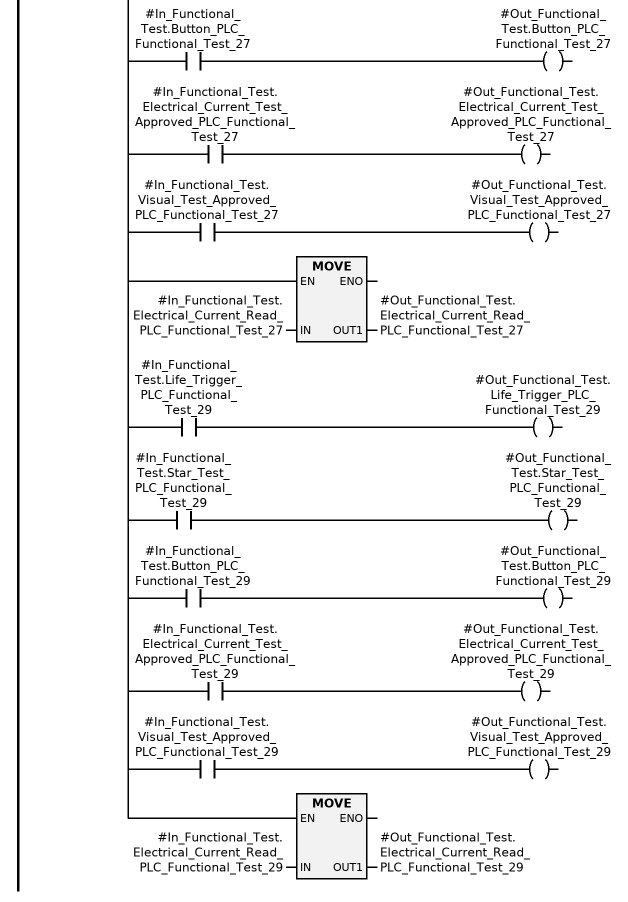
   RUNG wire#powerrail
      { S7_Templates := "SrcType := SInt" } EQ_Contact(in1 := #Test_Station, in2 := 13)
      wire#w1
      Contact( #Life_Trigger )
      Coil( #Out_Functional_Test.Life_Trigger_PLC_Functional_Test_13 )
   END_RUNG
   RUNG wire#w1
      Contact( #Star_Test )
      Coil( #Out_Functional_Test.Star_Test_PLC_Functional_Test_13 )
   END_RUNG
   RUNG wire#w1
      Contact( #Button_Start_Approve )
      Coil( #Out_Functional_Test.Button_PLC_Functional_Test_13 )
   END_RUNG
   RUNG wire#w1
      Contact( #Electrical_Current_Test_Approved )
      Coil( #Out_Functional_Test.Electrical_Current_Test_Approved_PLC_Functional_Test_13 )
   END_RUNG
   RUNG wire#w1
      Contact( #Visual_Test_Approved )
      Coil( #Out_Functional_Test.Visual_Test_Approved_PLC_Functional_Test_13 )
   END_RUNG
   RUNG wire#w1
      Contact( #In_Test_Parameters.Reset_PLC_Functional_Test_13 )
      Coil( #Reset_Functional_Test )
   END_RUNG
   RUNG wire#w1
      Move(in := #Electrical_Current_Read, out1 => #Out_Functional_Test.Electrical_Current_Read_PLC_Functional_Test_13)
   END_RUNG
   RUNG wire#w1
      Contact( #In_Functional_Test.Life_Trigger_PLC_Functional_Test_15 )
      Coil( #Out_Functional_Test.Life_Trigger_PLC_Functional_Test_15 )
   END_RUNG
   RUNG wire#w1
      Contact( #In_Functional_Test.Star_Test_PLC_Functional_Test_15 )
      Coil( #Out_Functional_Test.Star_Test_PLC_Functional_Test_15 )
   END_RUNG
   RUNG wire#w1
      Contact( #In_Functional_Test.Button_PLC_Functional_Test_15 )
      Coil( #Out_Functional_Test.Button_PLC_Functional_Test_15 )
   END_RUNG
   RUNG wire#w1
      Contact( #In_Functional_Test.Electrical_Current_Test_Approved_PLC_Functional_Test_15 )
      Coil( #Out_Functional_Test.Electrical_Current_Test_Approved_PLC_Functional_Test_15 )
   END_RUNG
   RUNG wire#w1
      Contact( #In_Functional_Test.Visual_Test_Approved_PLC_Functional_Test_15 )
      Coil( #Out_Functional_Test.Visual_Test_Approved_PLC_Functional_Test_15 )
   END_RUNG
   RUNG wire#w1
      Move(in := #In_Functional_Test.Electrical_Current_Read_PLC_Functional_Test_15, out1 => #Out_Functional_Test.Electrical_Current_Read_PLC_Functional_Test_15)
   END_RUNG
   RUNG wire#w1
      Contact( #In_Functional_Test.Life_Trigger_PLC_Functional_Test_17 )
      Coil( #Out_Functional_Test.Life_Trigger_PLC_Functional_Test_17 )
   END_RUNG
   RUNG wire#w1
      Contact( #In_Functional_Test.Star_Test_PLC_Functional_Test_17 )
      Coil( #Out_Functional_Test.Star_Test_PLC_Functional_Test_17 )
   END_RUNG
   RUNG wire#w1
      Contact( #In_Functional_Test.Button_PLC_Functional_Test_17 )
      Coil( #Out_Functional_Test.Button_PLC_Functional_Test_17 )
   END_RUNG
   RUNG wire#w1
      Contact( #In_Functional_Test.Electrical_Current_Test_Approved_PLC_Functional_Test_17 )
      Coil( #Out_Functional_Test.Electrical_Current_Test_Approved_PLC_Functional_Test_17 )
   END_RUNG
   RUNG wire#w1
      Contact( #In_Functional_Test.Visual_Test_Approved_PLC_Functional_Test_17 )
      Coil( #Out_Functional_Test.Visual_Test_Approved_PLC_Functional_Test_17 )
   END_RUNG
   RUNG wire#w1
      Move(in := #In_Functional_Test.Electrical_Current_Read_PLC_Functional_Test_17, out1 => #Out_Functional_Test.Electrical_Current_Read_PLC_Functional_Test_17)
   END_RUNG
   RUNG wire#w1
      Contact( #In_Functional_Test.Life_Trigger_PLC_Functional_Test_19 )
      Coil( #Out_Functional_Test.Life_Trigger_PLC_Functional_Test_19 )
   END_RUNG
   RUNG wire#w1
      Contact( #In_Functional_Test.Star_Test_PLC_Functional_Test_19 )
      Coil( #Out_Functional_Test.Star_Test_PLC_Functional_Test_19 )
   END_RUNG
   RUNG wire#w1
      Contact( #In_Functional_Test.Button_PLC_Functional_Test_19 )
      Coil( #Out_Functional_Test.Button_PLC_Functional_Test_19 )
   END_RUNG
   RUNG wire#w1
      Contact( #In_Functional_Test.Electrical_Current_Test_Approved_PLC_Functional_Test_19 )
      Coil( #Out_Functional_Test.Electrical_Current_Test_Approved_PLC_Functional_Test_19 )
   END_RUNG
   RUNG wire#w1
      Contact( #In_Functional_Test.Visual_Test_Approved_PLC_Functional_Test_19 )
      Coil( #Out_Functional_Test.Visual_Test_Approved_PLC_Functional_Test_19 )
   END_RUNG
   RUNG wire#w1
      Move(in := #In_Functional_Test.Electrical_Current_Read_PLC_Functional_Test_19, out1 => #Out_Functional_Test.Electrical_Current_Read_PLC_Functional_Test_19)
   END_RUNG
   RUNG wire#w1
      Contact( #In_Functional_Test.Life_Trigger_PLC_Functional_Test_21 )
      Coil( #Out_Functional_Test.Life_Trigger_PLC_Functional_Test_21 )
   END_RUNG
   RUNG wire#w1
      Contact( #In_Functional_Test.Star_Test_PLC_Functional_Test_21 )
      Coil( #Out_Functional_Test.Star_Test_PLC_Functional_Test_21 )
   END_RUNG
   RUNG wire#w1
      Contact( #In_Functional_Test.Button_PLC_Functional_Test_21 )
      Coil( #Out_Functional_Test.Button_PLC_Functional_Test_21 )
   END_RUNG
   RUNG wire#w1
      Contact( #In_Functional_Test.Electrical_Current_Test_Approved_PLC_Functional_Test_21 )
      Coil( #Out_Functional_Test.Electrical_Current_Test_Approved_PLC_Functional_Test_21 )
   END_RUNG
   RUNG wire#w1
      Contact( #In_Functional_Test.Visual_Test_Approved_PLC_Functional_Test_21 )
      Coil( #Out_Functional_Test.Visual_Test_Approved_PLC_Functional_Test_21 )
   END_RUNG
   RUNG wire#w1
      Move(in := #In_Functional_Test.Electrical_Current_Read_PLC_Functional_Test_21, out1 => #Out_Functional_Test.Electrical_Current_Read_PLC_Functional_Test_21)
   END_RUNG
   RUNG wire#w1
      Contact( #In_Functional_Test.Life_Trigger_PLC_Functional_Test_23 )
      Coil( #Out_Functional_Test.Life_Trigger_PLC_Functional_Test_23 )
   END_RUNG
   RUNG wire#w1
      Contact( #In_Functional_Test.Star_Test_PLC_Functional_Test_23 )
      Coil( #Out_Functional_Test.Star_Test_PLC_Functional_Test_23 )
   END_RUNG
   RUNG wire#w1
      Contact( #In_Functional_Test.Button_PLC_Functional_Test_23 )
      Coil( #Out_Functional_Test.Button_PLC_Functional_Test_23 )
   END_RUNG
   RUNG wire#w1
      Contact( #In_Functional_Test.Electrical_Current_Test_Approved_PLC_Functional_Test_23 )
      Coil( #Out_Functional_Test.Electrical_Current_Test_Approved_PLC_Functional_Test_23 )
   END_RUNG
   RUNG wire#w1
      Contact( #In_Functional_Test.Visual_Test_Approved_PLC_Functional_Test_23 )
      Coil( #Out_Functional_Test.Visual_Test_Approved_PLC_Functional_Test_23 )
   END_RUNG
   RUNG wire#w1
      Move(in := #In_Functional_Test.Electrical_Current_Read_PLC_Functional_Test_23, out1 => #Out_Functional_Test.Electrical_Current_Read_PLC_Functional_Test_23)
   END_RUNG
   RUNG wire#w1
      Contact( #In_Functional_Test.Life_Trigger_PLC_Functional_Test_25 )
      Coil( #Out_Functional_Test.Life_Trigger_PLC_Functional_Test_25 )
   END_RUNG
   RUNG wire#w1
      Contact( #In_Functional_Test.Star_Test_PLC_Functional_Test_25 )
      Coil( #Out_Functional_Test.Star_Test_PLC_Functional_Test_25 )
   END_RUNG
   RUNG wire#w1
      Contact( #In_Functional_Test.Button_PLC_Functional_Test_25 )
      Coil( #Out_Functional_Test.Button_PLC_Functional_Test_25 )
   END_RUNG
   RUNG wire#w1
      Contact( #In_Functional_Test.Electrical_Current_Test_Approved_PLC_Functional_Test_25 )
      Coil( #Out_Functional_Test.Electrical_Current_Test_Approved_PLC_Functional_Test_25 )
   END_RUNG
   RUNG wire#w1
      Contact( #In_Functional_Test.Visual_Test_Approved_PLC_Functional_Test_25 )
      Coil( #Out_Functional_Test.Visual_Test_Approved_PLC_Functional_Test_25 )
   END_RUNG
   RUNG wire#w1
      Move(in := #In_Functional_Test.Electrical_Current_Read_PLC_Functional_Test_25, out1 => #Out_Functional_Test.Electrical_Current_Read_PLC_Functional_Test_25)
   END_RUNG
   RUNG wire#w1
      Contact( #In_Functional_Test.Life_Trigger_PLC_Functional_Test_27 )
      Coil( #Out_Functional_Test.Life_Trigger_PLC_Functional_Test_27 )
   END_RUNG
   RUNG wire#w1
      Contact( #In_Functional_Test.Star_Test_PLC_Functional_Test_27 )
      Coil( #Out_Functional_Test.Star_Test_PLC_Functional_Test_27 )
   END_RUNG
   RUNG wire#w1
      Contact( #In_Functional_Test.Button_PLC_Functional_Test_27 )
      Coil( #Out_Functional_Test.Button_PLC_Functional_Test_27 )
   END_RUNG
   RUNG wire#w1
      Contact( #In_Functional_Test.Electrical_Current_Test_Approved_PLC_Functional_Test_27 )
      Coil( #Out_Functional_Test.Electrical_Current_Test_Approved_PLC_Functional_Test_27 )
   END_RUNG
   RUNG wire#w1
      Contact( #In_Functional_Test.Visual_Test_Approved_PLC_Functional_Test_27 )
      Coil( #Out_Functional_Test.Visual_Test_Approved_PLC_Functional_Test_27 )
   END_RUNG
   RUNG wire#w1
      Move(in := #In_Functional_Test.Electrical_Current_Read_PLC_Functional_Test_27, out1 => #Out_Functional_Test.Electrical_Current_Read_PLC_Functional_Test_27)
   END_RUNG
   RUNG wire#w1
      Contact( #In_Functional_Test.Life_Trigger_PLC_Functional_Test_29 )
      Coil( #Out_Functional_Test.Life_Trigger_PLC_Functional_Test_29 )
   END_RUNG
   RUNG wire#w1
      Contact( #In_Functional_Test.Star_Test_PLC_Functional_Test_29 )
      Coil( #Out_Functional_Test.Star_Test_PLC_Functional_Test_29 )
   END_RUNG
   RUNG wire#w1
      Contact( #In_Functional_Test.Button_PLC_Functional_Test_29 )
      Coil( #Out_Functional_Test.Button_PLC_Functional_Test_29 )
   END_RUNG
   RUNG wire#w1
      Contact( #In_Functional_Test.Electrical_Current_Test_Approved_PLC_Functional_Test_29 )
      Coil( #Out_Functional_Test.Electrical_Current_Test_Approved_PLC_Functional_Test_29 )
   END_RUNG
   RUNG wire#w1
      Contact( #In_Functional_Test.Visual_Test_Approved_PLC_Functional_Test_29 )
      Coil( #Out_Functional_Test.Visual_Test_Approved_PLC_Functional_Test_29 )
   END_RUNG
   RUNG wire#w1
      Move(in := #In_Functional_Test.Electrical_Current_Read_PLC_Functional_Test_29, out1 => #Out_Functional_Test.Electrical_Current_Read_PLC_Functional_Test_29)
   END_RUNG
   // the same network as SCL:
   #_w1 := #Test_Station = 13;
   #Out_Functional_Test.Life_Trigger_PLC_Functional_Test_13 := #_w1 AND #Life_Trigger;
   #Out_Functional_Test.Star_Test_PLC_Functional_Test_13 := #_w1 AND #Star_Test;
   #Out_Functional_Test.Button_PLC_Functional_Test_13 := #_w1 AND #Button_Start_Approve;
   #Out_Functional_Test.Electrical_Current_Test_Approved_PLC_Functional_Test_13 := #_w1 AND #Electrical_Current_Test_Approved;
   #Out_Functional_Test.Visual_Test_Approved_PLC_Functional_Test_13 := #_w1 AND #Visual_Test_Approved;
   #Reset_Functional_Test := #_w1 AND #In_Test_Parameters.Reset_PLC_Functional_Test_13;
   IF #_w1 THEN
       #Out_Functional_Test.Electrical_Current_Read_PLC_Functional_Test_13 := #Electrical_Current_Read;
   END_IF;
   #Out_Functional_Test.Life_Trigger_PLC_Functional_Test_15 := #_w1 AND #In_Functional_Test.Life_Trigger_PLC_Functional_Test_15;
   #Out_Functional_Test.Star_Test_PLC_Functional_Test_15 := #_w1 AND #In_Functional_Test.Star_Test_PLC_Functional_Test_15;
   #Out_Functional_Test.Button_PLC_Functional_Test_15 := #_w1 AND #In_Functional_Test.Button_PLC_Functional_Test_15;
   #Out_Functional_Test.Electrical_Current_Test_Approved_PLC_Functional_Test_15 := #_w1 AND #In_Functional_Test.Electrical_Current_Test_Approved_PLC_Functional_Test_15;
   #Out_Functional_Test.Visual_Test_Approved_PLC_Functional_Test_15 := #_w1 AND #In_Functional_Test.Visual_Test_Approved_PLC_Functional_Test_15;
   IF #_w1 THEN
       #Out_Functional_Test.Electrical_Current_Read_PLC_Functional_Test_15 := #In_Functional_Test.Electrical_Current_Read_PLC_Functional_Test_15;
   END_IF;
   #Out_Functional_Test.Life_Trigger_PLC_Functional_Test_17 := #_w1 AND #In_Functional_Test.Life_Trigger_PLC_Functional_Test_17;
   #Out_Functional_Test.Star_Test_PLC_Functional_Test_17 := #_w1 AND #In_Functional_Test.Star_Test_PLC_Functional_Test_17;
   #Out_Functional_Test.Button_PLC_Functional_Test_17 := #_w1 AND #In_Functional_Test.Button_PLC_Functional_Test_17;
   #Out_Functional_Test.Electrical_Current_Test_Approved_PLC_Functional_Test_17 := #_w1 AND #In_Functional_Test.Electrical_Current_Test_Approved_PLC_Functional_Test_17;
   #Out_Functional_Test.Visual_Test_Approved_PLC_Functional_Test_17 := #_w1 AND #In_Functional_Test.Visual_Test_Approved_PLC_Functional_Test_17;
   IF #_w1 THEN
       #Out_Functional_Test.Electrical_Current_Read_PLC_Functional_Test_17 := #In_Functional_Test.Electrical_Current_Read_PLC_Functional_Test_17;
   END_IF;
   #Out_Functional_Test.Life_Trigger_PLC_Functional_Test_19 := #_w1 AND #In_Functional_Test.Life_Trigger_PLC_Functional_Test_19;
   #Out_Functional_Test.Star_Test_PLC_Functional_Test_19 := #_w1 AND #In_Functional_Test.Star_Test_PLC_Functional_Test_19;
   #Out_Functional_Test.Button_PLC_Functional_Test_19 := #_w1 AND #In_Functional_Test.Button_PLC_Functional_Test_19;
   #Out_Functional_Test.Electrical_Current_Test_Approved_PLC_Functional_Test_19 := #_w1 AND #In_Functional_Test.Electrical_Current_Test_Approved_PLC_Functional_Test_19;
   #Out_Functional_Test.Visual_Test_Approved_PLC_Functional_Test_19 := #_w1 AND #In_Functional_Test.Visual_Test_Approved_PLC_Functional_Test_19;
   IF #_w1 THEN
       #Out_Functional_Test.Electrical_Current_Read_PLC_Functional_Test_19 := #In_Functional_Test.Electrical_Current_Read_PLC_Functional_Test_19;
   END_IF;
   #Out_Functional_Test.Life_Trigger_PLC_Functional_Test_21 := #_w1 AND #In_Functional_Test.Life_Trigger_PLC_Functional_Test_21;
   #Out_Functional_Test.Star_Test_PLC_Functional_Test_21 := #_w1 AND #In_Functional_Test.Star_Test_PLC_Functional_Test_21;
   #Out_Functional_Test.Button_PLC_Functional_Test_21 := #_w1 AND #In_Functional_Test.Button_PLC_Functional_Test_21;
   #Out_Functional_Test.Electrical_Current_Test_Approved_PLC_Functional_Test_21 := #_w1 AND #In_Functional_Test.Electrical_Current_Test_Approved_PLC_Functional_Test_21;
   #Out_Functional_Test.Visual_Test_Approved_PLC_Functional_Test_21 := #_w1 AND #In_Functional_Test.Visual_Test_Approved_PLC_Functional_Test_21;
   IF #_w1 THEN
       #Out_Functional_Test.Electrical_Current_Read_PLC_Functional_Test_21 := #In_Functional_Test.Electrical_Current_Read_PLC_Functional_Test_21;
   END_IF;
   #Out_Functional_Test.Life_Trigger_PLC_Functional_Test_23 := #_w1 AND #In_Functional_Test.Life_Trigger_PLC_Functional_Test_23;
   #Out_Functional_Test.Star_Test_PLC_Functional_Test_23 := #_w1 AND #In_Functional_Test.Star_Test_PLC_Functional_Test_23;
   #Out_Functional_Test.Button_PLC_Functional_Test_23 := #_w1 AND #In_Functional_Test.Button_PLC_Functional_Test_23;
   #Out_Functional_Test.Electrical_Current_Test_Approved_PLC_Functional_Test_23 := #_w1 AND #In_Functional_Test.Electrical_Current_Test_Approved_PLC_Functional_Test_23;
   #Out_Functional_Test.Visual_Test_Approved_PLC_Functional_Test_23 := #_w1 AND #In_Functional_Test.Visual_Test_Approved_PLC_Functional_Test_23;
   IF #_w1 THEN
       #Out_Functional_Test.Electrical_Current_Read_PLC_Functional_Test_23 := #In_Functional_Test.Electrical_Current_Read_PLC_Functional_Test_23;
   END_IF;
   #Out_Functional_Test.Life_Trigger_PLC_Functional_Test_25 := #_w1 AND #In_Functional_Test.Life_Trigger_PLC_Functional_Test_25;
   #Out_Functional_Test.Star_Test_PLC_Functional_Test_25 := #_w1 AND #In_Functional_Test.Star_Test_PLC_Functional_Test_25;
   #Out_Functional_Test.Button_PLC_Functional_Test_25 := #_w1 AND #In_Functional_Test.Button_PLC_Functional_Test_25;
   #Out_Functional_Test.Electrical_Current_Test_Approved_PLC_Functional_Test_25 := #_w1 AND #In_Functional_Test.Electrical_Current_Test_Approved_PLC_Functional_Test_25;
   #Out_Functional_Test.Visual_Test_Approved_PLC_Functional_Test_25 := #_w1 AND #In_Functional_Test.Visual_Test_Approved_PLC_Functional_Test_25;
   IF #_w1 THEN
       #Out_Functional_Test.Electrical_Current_Read_PLC_Functional_Test_25 := #In_Functional_Test.Electrical_Current_Read_PLC_Functional_Test_25;
   END_IF;
   #Out_Functional_Test.Life_Trigger_PLC_Functional_Test_27 := #_w1 AND #In_Functional_Test.Life_Trigger_PLC_Functional_Test_27;
   #Out_Functional_Test.Star_Test_PLC_Functional_Test_27 := #_w1 AND #In_Functional_Test.Star_Test_PLC_Functional_Test_27;
   #Out_Functional_Test.Button_PLC_Functional_Test_27 := #_w1 AND #In_Functional_Test.Button_PLC_Functional_Test_27;
   #Out_Functional_Test.Electrical_Current_Test_Approved_PLC_Functional_Test_27 := #_w1 AND #In_Functional_Test.Electrical_Current_Test_Approved_PLC_Functional_Test_27;
   #Out_Functional_Test.Visual_Test_Approved_PLC_Functional_Test_27 := #_w1 AND #In_Functional_Test.Visual_Test_Approved_PLC_Functional_Test_27;
   IF #_w1 THEN
       #Out_Functional_Test.Electrical_Current_Read_PLC_Functional_Test_27 := #In_Functional_Test.Electrical_Current_Read_PLC_Functional_Test_27;
   END_IF;
   #Out_Functional_Test.Life_Trigger_PLC_Functional_Test_29 := #_w1 AND #In_Functional_Test.Life_Trigger_PLC_Functional_Test_29;
   #Out_Functional_Test.Star_Test_PLC_Functional_Test_29 := #_w1 AND #In_Functional_Test.Star_Test_PLC_Functional_Test_29;
   #Out_Functional_Test.Button_PLC_Functional_Test_29 := #_w1 AND #In_Functional_Test.Button_PLC_Functional_Test_29;
   #Out_Functional_Test.Electrical_Current_Test_Approved_PLC_Functional_Test_29 := #_w1 AND #In_Functional_Test.Electrical_Current_Test_Approved_PLC_Functional_Test_29;
   #Out_Functional_Test.Visual_Test_Approved_PLC_Functional_Test_29 := #_w1 AND #In_Functional_Test.Visual_Test_Approved_PLC_Functional_Test_29;
   IF #_w1 THEN
       #Out_Functional_Test.Electrical_Current_Read_PLC_Functional_Test_29 := #In_Functional_Test.Electrical_Current_Read_PLC_Functional_Test_29;
   END_IF;
END_REGION

REGION Network 9: Functional Test Station 15
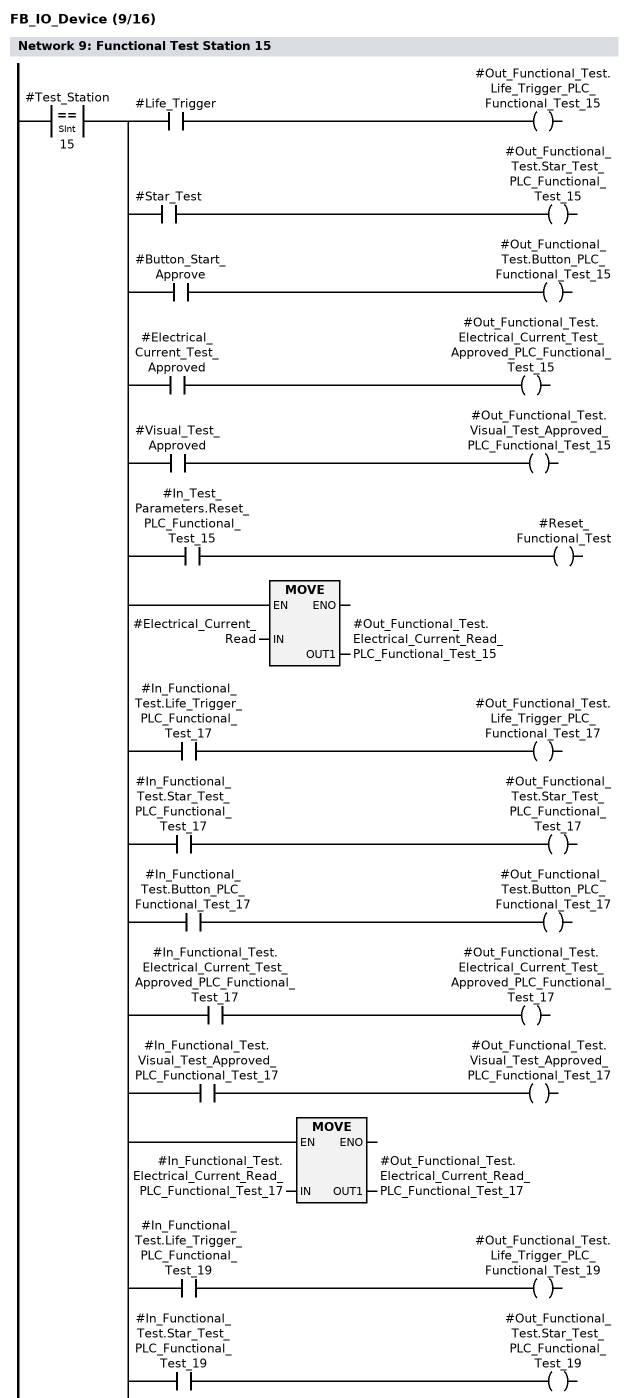
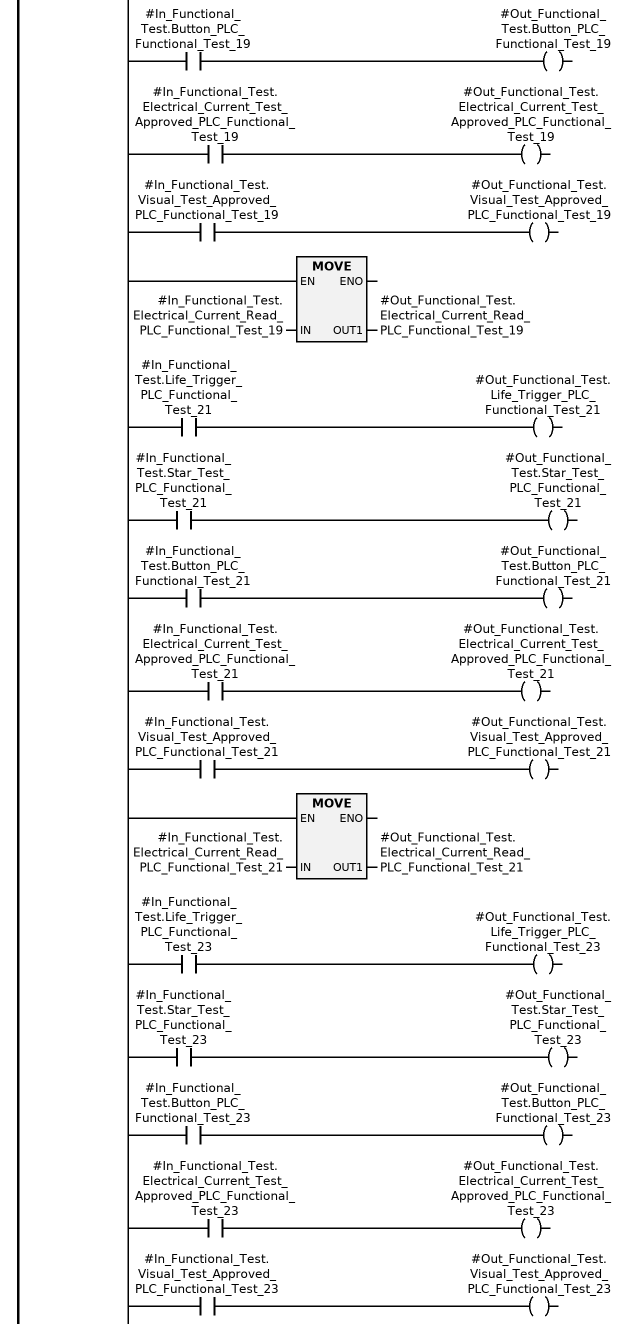
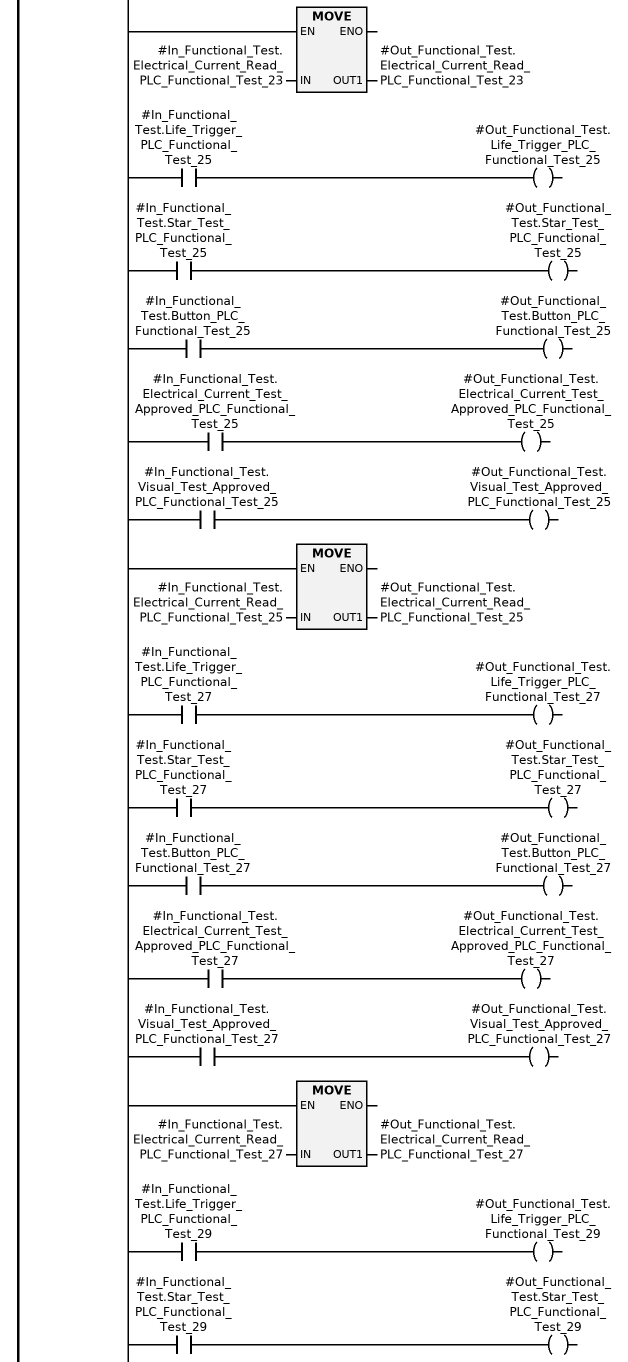
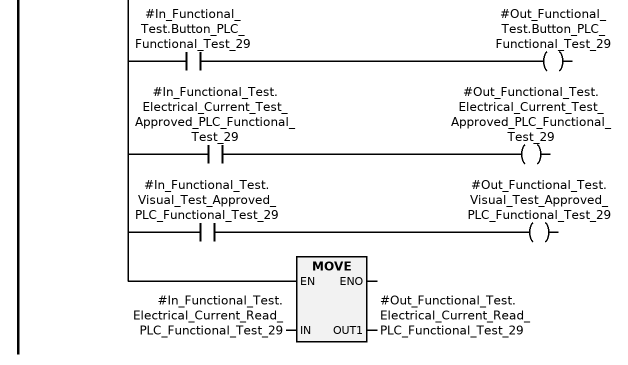
   RUNG wire#powerrail
      { S7_Templates := "SrcType := SInt" } EQ_Contact(in1 := #Test_Station, in2 := 15)
      wire#w1
      Contact( #Life_Trigger )
      Coil( #Out_Functional_Test.Life_Trigger_PLC_Functional_Test_15 )
   END_RUNG
   RUNG wire#w1
      Contact( #Star_Test )
      Coil( #Out_Functional_Test.Star_Test_PLC_Functional_Test_15 )
   END_RUNG
   RUNG wire#w1
      Contact( #Button_Start_Approve )
      Coil( #Out_Functional_Test.Button_PLC_Functional_Test_15 )
   END_RUNG
   RUNG wire#w1
      Contact( #Electrical_Current_Test_Approved )
      Coil( #Out_Functional_Test.Electrical_Current_Test_Approved_PLC_Functional_Test_15 )
   END_RUNG
   RUNG wire#w1
      Contact( #Visual_Test_Approved )
      Coil( #Out_Functional_Test.Visual_Test_Approved_PLC_Functional_Test_15 )
   END_RUNG
   RUNG wire#w1
      Contact( #In_Test_Parameters.Reset_PLC_Functional_Test_15 )
      Coil( #Reset_Functional_Test )
   END_RUNG
   RUNG wire#w1
      Move(in := #Electrical_Current_Read, out1 => #Out_Functional_Test.Electrical_Current_Read_PLC_Functional_Test_15)
   END_RUNG
   RUNG wire#w1
      Contact( #In_Functional_Test.Life_Trigger_PLC_Functional_Test_17 )
      Coil( #Out_Functional_Test.Life_Trigger_PLC_Functional_Test_17 )
   END_RUNG
   RUNG wire#w1
      Contact( #In_Functional_Test.Star_Test_PLC_Functional_Test_17 )
      Coil( #Out_Functional_Test.Star_Test_PLC_Functional_Test_17 )
   END_RUNG
   RUNG wire#w1
      Contact( #In_Functional_Test.Button_PLC_Functional_Test_17 )
      Coil( #Out_Functional_Test.Button_PLC_Functional_Test_17 )
   END_RUNG
   RUNG wire#w1
      Contact( #In_Functional_Test.Electrical_Current_Test_Approved_PLC_Functional_Test_17 )
      Coil( #Out_Functional_Test.Electrical_Current_Test_Approved_PLC_Functional_Test_17 )
   END_RUNG
   RUNG wire#w1
      Contact( #In_Functional_Test.Visual_Test_Approved_PLC_Functional_Test_17 )
      Coil( #Out_Functional_Test.Visual_Test_Approved_PLC_Functional_Test_17 )
   END_RUNG
   RUNG wire#w1
      Move(in := #In_Functional_Test.Electrical_Current_Read_PLC_Functional_Test_17, out1 => #Out_Functional_Test.Electrical_Current_Read_PLC_Functional_Test_17)
   END_RUNG
   RUNG wire#w1
      Contact( #In_Functional_Test.Life_Trigger_PLC_Functional_Test_19 )
      Coil( #Out_Functional_Test.Life_Trigger_PLC_Functional_Test_19 )
   END_RUNG
   RUNG wire#w1
      Contact( #In_Functional_Test.Star_Test_PLC_Functional_Test_19 )
      Coil( #Out_Functional_Test.Star_Test_PLC_Functional_Test_19 )
   END_RUNG
   RUNG wire#w1
      Contact( #In_Functional_Test.Button_PLC_Functional_Test_19 )
      Coil( #Out_Functional_Test.Button_PLC_Functional_Test_19 )
   END_RUNG
   RUNG wire#w1
      Contact( #In_Functional_Test.Electrical_Current_Test_Approved_PLC_Functional_Test_19 )
      Coil( #Out_Functional_Test.Electrical_Current_Test_Approved_PLC_Functional_Test_19 )
   END_RUNG
   RUNG wire#w1
      Contact( #In_Functional_Test.Visual_Test_Approved_PLC_Functional_Test_19 )
      Coil( #Out_Functional_Test.Visual_Test_Approved_PLC_Functional_Test_19 )
   END_RUNG
   RUNG wire#w1
      Move(in := #In_Functional_Test.Electrical_Current_Read_PLC_Functional_Test_19, out1 => #Out_Functional_Test.Electrical_Current_Read_PLC_Functional_Test_19)
   END_RUNG
   RUNG wire#w1
      Contact( #In_Functional_Test.Life_Trigger_PLC_Functional_Test_21 )
      Coil( #Out_Functional_Test.Life_Trigger_PLC_Functional_Test_21 )
   END_RUNG
   RUNG wire#w1
      Contact( #In_Functional_Test.Star_Test_PLC_Functional_Test_21 )
      Coil( #Out_Functional_Test.Star_Test_PLC_Functional_Test_21 )
   END_RUNG
   RUNG wire#w1
      Contact( #In_Functional_Test.Button_PLC_Functional_Test_21 )
      Coil( #Out_Functional_Test.Button_PLC_Functional_Test_21 )
   END_RUNG
   RUNG wire#w1
      Contact( #In_Functional_Test.Electrical_Current_Test_Approved_PLC_Functional_Test_21 )
      Coil( #Out_Functional_Test.Electrical_Current_Test_Approved_PLC_Functional_Test_21 )
   END_RUNG
   RUNG wire#w1
      Contact( #In_Functional_Test.Visual_Test_Approved_PLC_Functional_Test_21 )
      Coil( #Out_Functional_Test.Visual_Test_Approved_PLC_Functional_Test_21 )
   END_RUNG
   RUNG wire#w1
      Move(in := #In_Functional_Test.Electrical_Current_Read_PLC_Functional_Test_21, out1 => #Out_Functional_Test.Electrical_Current_Read_PLC_Functional_Test_21)
   END_RUNG
   RUNG wire#w1
      Contact( #In_Functional_Test.Life_Trigger_PLC_Functional_Test_23 )
      Coil( #Out_Functional_Test.Life_Trigger_PLC_Functional_Test_23 )
   END_RUNG
   RUNG wire#w1
      Contact( #In_Functional_Test.Star_Test_PLC_Functional_Test_23 )
      Coil( #Out_Functional_Test.Star_Test_PLC_Functional_Test_23 )
   END_RUNG
   RUNG wire#w1
      Contact( #In_Functional_Test.Button_PLC_Functional_Test_23 )
      Coil( #Out_Functional_Test.Button_PLC_Functional_Test_23 )
   END_RUNG
   RUNG wire#w1
      Contact( #In_Functional_Test.Electrical_Current_Test_Approved_PLC_Functional_Test_23 )
      Coil( #Out_Functional_Test.Electrical_Current_Test_Approved_PLC_Functional_Test_23 )
   END_RUNG
   RUNG wire#w1
      Contact( #In_Functional_Test.Visual_Test_Approved_PLC_Functional_Test_23 )
      Coil( #Out_Functional_Test.Visual_Test_Approved_PLC_Functional_Test_23 )
   END_RUNG
   RUNG wire#w1
      Move(in := #In_Functional_Test.Electrical_Current_Read_PLC_Functional_Test_23, out1 => #Out_Functional_Test.Electrical_Current_Read_PLC_Functional_Test_23)
   END_RUNG
   RUNG wire#w1
      Contact( #In_Functional_Test.Life_Trigger_PLC_Functional_Test_25 )
      Coil( #Out_Functional_Test.Life_Trigger_PLC_Functional_Test_25 )
   END_RUNG
   RUNG wire#w1
      Contact( #In_Functional_Test.Star_Test_PLC_Functional_Test_25 )
      Coil( #Out_Functional_Test.Star_Test_PLC_Functional_Test_25 )
   END_RUNG
   RUNG wire#w1
      Contact( #In_Functional_Test.Button_PLC_Functional_Test_25 )
      Coil( #Out_Functional_Test.Button_PLC_Functional_Test_25 )
   END_RUNG
   RUNG wire#w1
      Contact( #In_Functional_Test.Electrical_Current_Test_Approved_PLC_Functional_Test_25 )
      Coil( #Out_Functional_Test.Electrical_Current_Test_Approved_PLC_Functional_Test_25 )
   END_RUNG
   RUNG wire#w1
      Contact( #In_Functional_Test.Visual_Test_Approved_PLC_Functional_Test_25 )
      Coil( #Out_Functional_Test.Visual_Test_Approved_PLC_Functional_Test_25 )
   END_RUNG
   RUNG wire#w1
      Move(in := #In_Functional_Test.Electrical_Current_Read_PLC_Functional_Test_25, out1 => #Out_Functional_Test.Electrical_Current_Read_PLC_Functional_Test_25)
   END_RUNG
   RUNG wire#w1
      Contact( #In_Functional_Test.Life_Trigger_PLC_Functional_Test_27 )
      Coil( #Out_Functional_Test.Life_Trigger_PLC_Functional_Test_27 )
   END_RUNG
   RUNG wire#w1
      Contact( #In_Functional_Test.Star_Test_PLC_Functional_Test_27 )
      Coil( #Out_Functional_Test.Star_Test_PLC_Functional_Test_27 )
   END_RUNG
   RUNG wire#w1
      Contact( #In_Functional_Test.Button_PLC_Functional_Test_27 )
      Coil( #Out_Functional_Test.Button_PLC_Functional_Test_27 )
   END_RUNG
   RUNG wire#w1
      Contact( #In_Functional_Test.Electrical_Current_Test_Approved_PLC_Functional_Test_27 )
      Coil( #Out_Functional_Test.Electrical_Current_Test_Approved_PLC_Functional_Test_27 )
   END_RUNG
   RUNG wire#w1
      Contact( #In_Functional_Test.Visual_Test_Approved_PLC_Functional_Test_27 )
      Coil( #Out_Functional_Test.Visual_Test_Approved_PLC_Functional_Test_27 )
   END_RUNG
   RUNG wire#w1
      Move(in := #In_Functional_Test.Electrical_Current_Read_PLC_Functional_Test_27, out1 => #Out_Functional_Test.Electrical_Current_Read_PLC_Functional_Test_27)
   END_RUNG
   RUNG wire#w1
      Contact( #In_Functional_Test.Life_Trigger_PLC_Functional_Test_29 )
      Coil( #Out_Functional_Test.Life_Trigger_PLC_Functional_Test_29 )
   END_RUNG
   RUNG wire#w1
      Contact( #In_Functional_Test.Star_Test_PLC_Functional_Test_29 )
      Coil( #Out_Functional_Test.Star_Test_PLC_Functional_Test_29 )
   END_RUNG
   RUNG wire#w1
      Contact( #In_Functional_Test.Button_PLC_Functional_Test_29 )
      Coil( #Out_Functional_Test.Button_PLC_Functional_Test_29 )
   END_RUNG
   RUNG wire#w1
      Contact( #In_Functional_Test.Electrical_Current_Test_Approved_PLC_Functional_Test_29 )
      Coil( #Out_Functional_Test.Electrical_Current_Test_Approved_PLC_Functional_Test_29 )
   END_RUNG
   RUNG wire#w1
      Contact( #In_Functional_Test.Visual_Test_Approved_PLC_Functional_Test_29 )
      Coil( #Out_Functional_Test.Visual_Test_Approved_PLC_Functional_Test_29 )
   END_RUNG
   RUNG wire#w1
      Move(in := #In_Functional_Test.Electrical_Current_Read_PLC_Functional_Test_29, out1 => #Out_Functional_Test.Electrical_Current_Read_PLC_Functional_Test_29)
   END_RUNG
   // the same network as SCL:
   #_w1 := #Test_Station = 15;
   #Out_Functional_Test.Life_Trigger_PLC_Functional_Test_15 := #_w1 AND #Life_Trigger;
   #Out_Functional_Test.Star_Test_PLC_Functional_Test_15 := #_w1 AND #Star_Test;
   #Out_Functional_Test.Button_PLC_Functional_Test_15 := #_w1 AND #Button_Start_Approve;
   #Out_Functional_Test.Electrical_Current_Test_Approved_PLC_Functional_Test_15 := #_w1 AND #Electrical_Current_Test_Approved;
   #Out_Functional_Test.Visual_Test_Approved_PLC_Functional_Test_15 := #_w1 AND #Visual_Test_Approved;
   #Reset_Functional_Test := #_w1 AND #In_Test_Parameters.Reset_PLC_Functional_Test_15;
   IF #_w1 THEN
       #Out_Functional_Test.Electrical_Current_Read_PLC_Functional_Test_15 := #Electrical_Current_Read;
   END_IF;
   #Out_Functional_Test.Life_Trigger_PLC_Functional_Test_17 := #_w1 AND #In_Functional_Test.Life_Trigger_PLC_Functional_Test_17;
   #Out_Functional_Test.Star_Test_PLC_Functional_Test_17 := #_w1 AND #In_Functional_Test.Star_Test_PLC_Functional_Test_17;
   #Out_Functional_Test.Button_PLC_Functional_Test_17 := #_w1 AND #In_Functional_Test.Button_PLC_Functional_Test_17;
   #Out_Functional_Test.Electrical_Current_Test_Approved_PLC_Functional_Test_17 := #_w1 AND #In_Functional_Test.Electrical_Current_Test_Approved_PLC_Functional_Test_17;
   #Out_Functional_Test.Visual_Test_Approved_PLC_Functional_Test_17 := #_w1 AND #In_Functional_Test.Visual_Test_Approved_PLC_Functional_Test_17;
   IF #_w1 THEN
       #Out_Functional_Test.Electrical_Current_Read_PLC_Functional_Test_17 := #In_Functional_Test.Electrical_Current_Read_PLC_Functional_Test_17;
   END_IF;
   #Out_Functional_Test.Life_Trigger_PLC_Functional_Test_19 := #_w1 AND #In_Functional_Test.Life_Trigger_PLC_Functional_Test_19;
   #Out_Functional_Test.Star_Test_PLC_Functional_Test_19 := #_w1 AND #In_Functional_Test.Star_Test_PLC_Functional_Test_19;
   #Out_Functional_Test.Button_PLC_Functional_Test_19 := #_w1 AND #In_Functional_Test.Button_PLC_Functional_Test_19;
   #Out_Functional_Test.Electrical_Current_Test_Approved_PLC_Functional_Test_19 := #_w1 AND #In_Functional_Test.Electrical_Current_Test_Approved_PLC_Functional_Test_19;
   #Out_Functional_Test.Visual_Test_Approved_PLC_Functional_Test_19 := #_w1 AND #In_Functional_Test.Visual_Test_Approved_PLC_Functional_Test_19;
   IF #_w1 THEN
       #Out_Functional_Test.Electrical_Current_Read_PLC_Functional_Test_19 := #In_Functional_Test.Electrical_Current_Read_PLC_Functional_Test_19;
   END_IF;
   #Out_Functional_Test.Life_Trigger_PLC_Functional_Test_21 := #_w1 AND #In_Functional_Test.Life_Trigger_PLC_Functional_Test_21;
   #Out_Functional_Test.Star_Test_PLC_Functional_Test_21 := #_w1 AND #In_Functional_Test.Star_Test_PLC_Functional_Test_21;
   #Out_Functional_Test.Button_PLC_Functional_Test_21 := #_w1 AND #In_Functional_Test.Button_PLC_Functional_Test_21;
   #Out_Functional_Test.Electrical_Current_Test_Approved_PLC_Functional_Test_21 := #_w1 AND #In_Functional_Test.Electrical_Current_Test_Approved_PLC_Functional_Test_21;
   #Out_Functional_Test.Visual_Test_Approved_PLC_Functional_Test_21 := #_w1 AND #In_Functional_Test.Visual_Test_Approved_PLC_Functional_Test_21;
   IF #_w1 THEN
       #Out_Functional_Test.Electrical_Current_Read_PLC_Functional_Test_21 := #In_Functional_Test.Electrical_Current_Read_PLC_Functional_Test_21;
   END_IF;
   #Out_Functional_Test.Life_Trigger_PLC_Functional_Test_23 := #_w1 AND #In_Functional_Test.Life_Trigger_PLC_Functional_Test_23;
   #Out_Functional_Test.Star_Test_PLC_Functional_Test_23 := #_w1 AND #In_Functional_Test.Star_Test_PLC_Functional_Test_23;
   #Out_Functional_Test.Button_PLC_Functional_Test_23 := #_w1 AND #In_Functional_Test.Button_PLC_Functional_Test_23;
   #Out_Functional_Test.Electrical_Current_Test_Approved_PLC_Functional_Test_23 := #_w1 AND #In_Functional_Test.Electrical_Current_Test_Approved_PLC_Functional_Test_23;
   #Out_Functional_Test.Visual_Test_Approved_PLC_Functional_Test_23 := #_w1 AND #In_Functional_Test.Visual_Test_Approved_PLC_Functional_Test_23;
   IF #_w1 THEN
       #Out_Functional_Test.Electrical_Current_Read_PLC_Functional_Test_23 := #In_Functional_Test.Electrical_Current_Read_PLC_Functional_Test_23;
   END_IF;
   #Out_Functional_Test.Life_Trigger_PLC_Functional_Test_25 := #_w1 AND #In_Functional_Test.Life_Trigger_PLC_Functional_Test_25;
   #Out_Functional_Test.Star_Test_PLC_Functional_Test_25 := #_w1 AND #In_Functional_Test.Star_Test_PLC_Functional_Test_25;
   #Out_Functional_Test.Button_PLC_Functional_Test_25 := #_w1 AND #In_Functional_Test.Button_PLC_Functional_Test_25;
   #Out_Functional_Test.Electrical_Current_Test_Approved_PLC_Functional_Test_25 := #_w1 AND #In_Functional_Test.Electrical_Current_Test_Approved_PLC_Functional_Test_25;
   #Out_Functional_Test.Visual_Test_Approved_PLC_Functional_Test_25 := #_w1 AND #In_Functional_Test.Visual_Test_Approved_PLC_Functional_Test_25;
   IF #_w1 THEN
       #Out_Functional_Test.Electrical_Current_Read_PLC_Functional_Test_25 := #In_Functional_Test.Electrical_Current_Read_PLC_Functional_Test_25;
   END_IF;
   #Out_Functional_Test.Life_Trigger_PLC_Functional_Test_27 := #_w1 AND #In_Functional_Test.Life_Trigger_PLC_Functional_Test_27;
   #Out_Functional_Test.Star_Test_PLC_Functional_Test_27 := #_w1 AND #In_Functional_Test.Star_Test_PLC_Functional_Test_27;
   #Out_Functional_Test.Button_PLC_Functional_Test_27 := #_w1 AND #In_Functional_Test.Button_PLC_Functional_Test_27;
   #Out_Functional_Test.Electrical_Current_Test_Approved_PLC_Functional_Test_27 := #_w1 AND #In_Functional_Test.Electrical_Current_Test_Approved_PLC_Functional_Test_27;
   #Out_Functional_Test.Visual_Test_Approved_PLC_Functional_Test_27 := #_w1 AND #In_Functional_Test.Visual_Test_Approved_PLC_Functional_Test_27;
   IF #_w1 THEN
       #Out_Functional_Test.Electrical_Current_Read_PLC_Functional_Test_27 := #In_Functional_Test.Electrical_Current_Read_PLC_Functional_Test_27;
   END_IF;
   #Out_Functional_Test.Life_Trigger_PLC_Functional_Test_29 := #_w1 AND #In_Functional_Test.Life_Trigger_PLC_Functional_Test_29;
   #Out_Functional_Test.Star_Test_PLC_Functional_Test_29 := #_w1 AND #In_Functional_Test.Star_Test_PLC_Functional_Test_29;
   #Out_Functional_Test.Button_PLC_Functional_Test_29 := #_w1 AND #In_Functional_Test.Button_PLC_Functional_Test_29;
   #Out_Functional_Test.Electrical_Current_Test_Approved_PLC_Functional_Test_29 := #_w1 AND #In_Functional_Test.Electrical_Current_Test_Approved_PLC_Functional_Test_29;
   #Out_Functional_Test.Visual_Test_Approved_PLC_Functional_Test_29 := #_w1 AND #In_Functional_Test.Visual_Test_Approved_PLC_Functional_Test_29;
   IF #_w1 THEN
       #Out_Functional_Test.Electrical_Current_Read_PLC_Functional_Test_29 := #In_Functional_Test.Electrical_Current_Read_PLC_Functional_Test_29;
   END_IF;
END_REGION

REGION Network 10: Functional Test Station 17
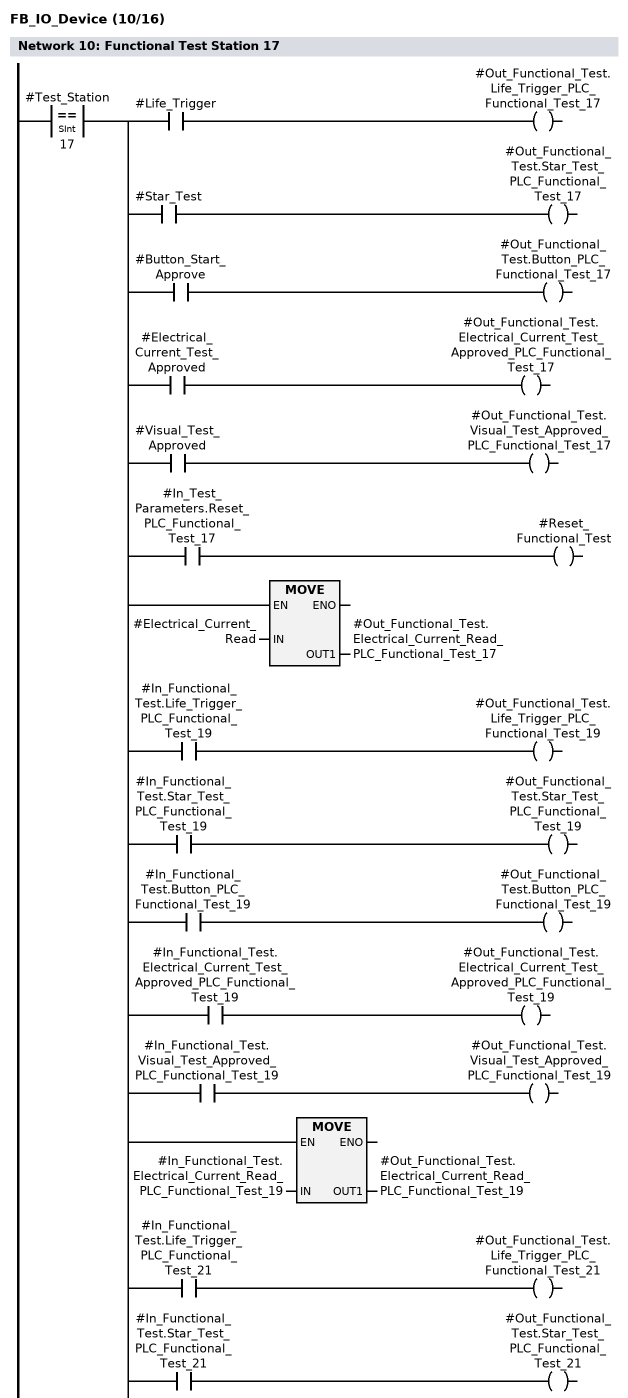
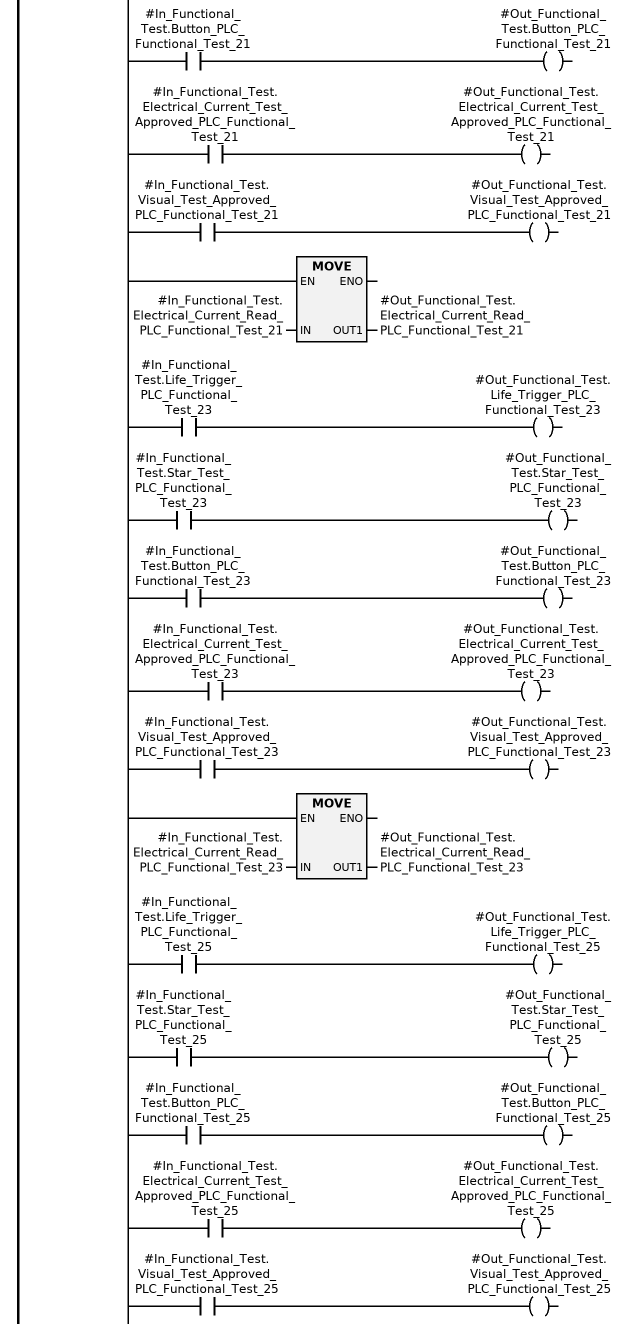
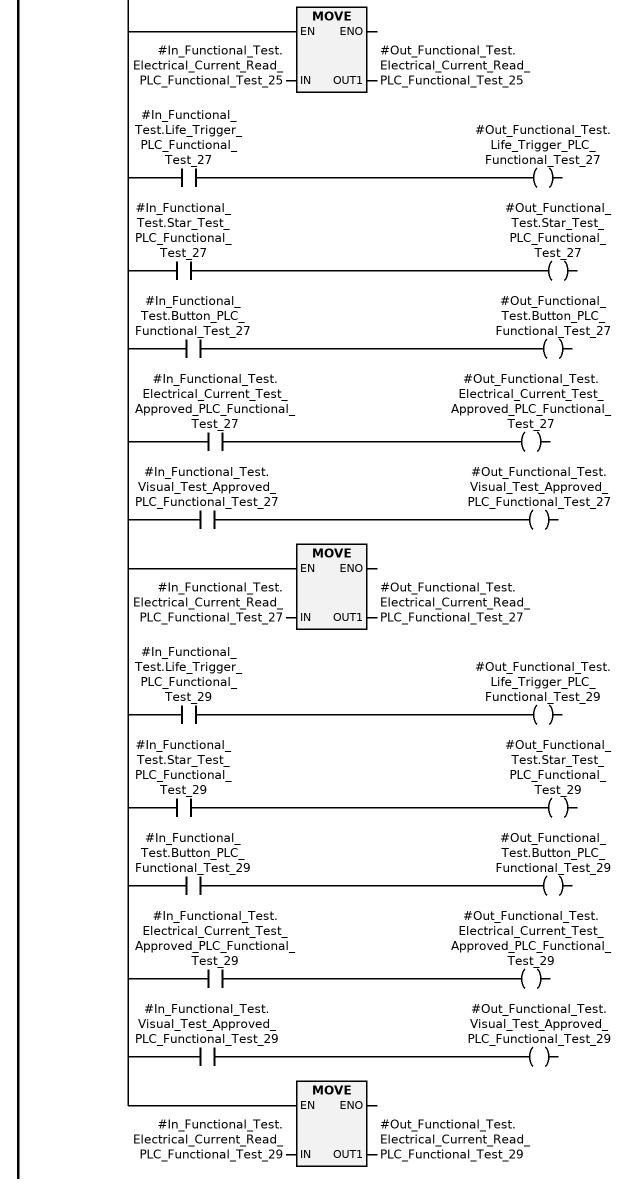
   RUNG wire#powerrail
      { S7_Templates := "SrcType := SInt" } EQ_Contact(in1 := #Test_Station, in2 := 17)
      wire#w1
      Contact( #Life_Trigger )
      Coil( #Out_Functional_Test.Life_Trigger_PLC_Functional_Test_17 )
   END_RUNG
   RUNG wire#w1
      Contact( #Star_Test )
      Coil( #Out_Functional_Test.Star_Test_PLC_Functional_Test_17 )
   END_RUNG
   RUNG wire#w1
      Contact( #Button_Start_Approve )
      Coil( #Out_Functional_Test.Button_PLC_Functional_Test_17 )
   END_RUNG
   RUNG wire#w1
      Contact( #Electrical_Current_Test_Approved )
      Coil( #Out_Functional_Test.Electrical_Current_Test_Approved_PLC_Functional_Test_17 )
   END_RUNG
   RUNG wire#w1
      Contact( #Visual_Test_Approved )
      Coil( #Out_Functional_Test.Visual_Test_Approved_PLC_Functional_Test_17 )
   END_RUNG
   RUNG wire#w1
      Contact( #In_Test_Parameters.Reset_PLC_Functional_Test_17 )
      Coil( #Reset_Functional_Test )
   END_RUNG
   RUNG wire#w1
      Move(in := #Electrical_Current_Read, out1 => #Out_Functional_Test.Electrical_Current_Read_PLC_Functional_Test_17)
   END_RUNG
   RUNG wire#w1
      Contact( #In_Functional_Test.Life_Trigger_PLC_Functional_Test_19 )
      Coil( #Out_Functional_Test.Life_Trigger_PLC_Functional_Test_19 )
   END_RUNG
   RUNG wire#w1
      Contact( #In_Functional_Test.Star_Test_PLC_Functional_Test_19 )
      Coil( #Out_Functional_Test.Star_Test_PLC_Functional_Test_19 )
   END_RUNG
   RUNG wire#w1
      Contact( #In_Functional_Test.Button_PLC_Functional_Test_19 )
      Coil( #Out_Functional_Test.Button_PLC_Functional_Test_19 )
   END_RUNG
   RUNG wire#w1
      Contact( #In_Functional_Test.Electrical_Current_Test_Approved_PLC_Functional_Test_19 )
      Coil( #Out_Functional_Test.Electrical_Current_Test_Approved_PLC_Functional_Test_19 )
   END_RUNG
   RUNG wire#w1
      Contact( #In_Functional_Test.Visual_Test_Approved_PLC_Functional_Test_19 )
      Coil( #Out_Functional_Test.Visual_Test_Approved_PLC_Functional_Test_19 )
   END_RUNG
   RUNG wire#w1
      Move(in := #In_Functional_Test.Electrical_Current_Read_PLC_Functional_Test_19, out1 => #Out_Functional_Test.Electrical_Current_Read_PLC_Functional_Test_19)
   END_RUNG
   RUNG wire#w1
      Contact( #In_Functional_Test.Life_Trigger_PLC_Functional_Test_21 )
      Coil( #Out_Functional_Test.Life_Trigger_PLC_Functional_Test_21 )
   END_RUNG
   RUNG wire#w1
      Contact( #In_Functional_Test.Star_Test_PLC_Functional_Test_21 )
      Coil( #Out_Functional_Test.Star_Test_PLC_Functional_Test_21 )
   END_RUNG
   RUNG wire#w1
      Contact( #In_Functional_Test.Button_PLC_Functional_Test_21 )
      Coil( #Out_Functional_Test.Button_PLC_Functional_Test_21 )
   END_RUNG
   RUNG wire#w1
      Contact( #In_Functional_Test.Electrical_Current_Test_Approved_PLC_Functional_Test_21 )
      Coil( #Out_Functional_Test.Electrical_Current_Test_Approved_PLC_Functional_Test_21 )
   END_RUNG
   RUNG wire#w1
      Contact( #In_Functional_Test.Visual_Test_Approved_PLC_Functional_Test_21 )
      Coil( #Out_Functional_Test.Visual_Test_Approved_PLC_Functional_Test_21 )
   END_RUNG
   RUNG wire#w1
      Move(in := #In_Functional_Test.Electrical_Current_Read_PLC_Functional_Test_21, out1 => #Out_Functional_Test.Electrical_Current_Read_PLC_Functional_Test_21)
   END_RUNG
   RUNG wire#w1
      Contact( #In_Functional_Test.Life_Trigger_PLC_Functional_Test_23 )
      Coil( #Out_Functional_Test.Life_Trigger_PLC_Functional_Test_23 )
   END_RUNG
   RUNG wire#w1
      Contact( #In_Functional_Test.Star_Test_PLC_Functional_Test_23 )
      Coil( #Out_Functional_Test.Star_Test_PLC_Functional_Test_23 )
   END_RUNG
   RUNG wire#w1
      Contact( #In_Functional_Test.Button_PLC_Functional_Test_23 )
      Coil( #Out_Functional_Test.Button_PLC_Functional_Test_23 )
   END_RUNG
   RUNG wire#w1
      Contact( #In_Functional_Test.Electrical_Current_Test_Approved_PLC_Functional_Test_23 )
      Coil( #Out_Functional_Test.Electrical_Current_Test_Approved_PLC_Functional_Test_23 )
   END_RUNG
   RUNG wire#w1
      Contact( #In_Functional_Test.Visual_Test_Approved_PLC_Functional_Test_23 )
      Coil( #Out_Functional_Test.Visual_Test_Approved_PLC_Functional_Test_23 )
   END_RUNG
   RUNG wire#w1
      Move(in := #In_Functional_Test.Electrical_Current_Read_PLC_Functional_Test_23, out1 => #Out_Functional_Test.Electrical_Current_Read_PLC_Functional_Test_23)
   END_RUNG
   RUNG wire#w1
      Contact( #In_Functional_Test.Life_Trigger_PLC_Functional_Test_25 )
      Coil( #Out_Functional_Test.Life_Trigger_PLC_Functional_Test_25 )
   END_RUNG
   RUNG wire#w1
      Contact( #In_Functional_Test.Star_Test_PLC_Functional_Test_25 )
      Coil( #Out_Functional_Test.Star_Test_PLC_Functional_Test_25 )
   END_RUNG
   RUNG wire#w1
      Contact( #In_Functional_Test.Button_PLC_Functional_Test_25 )
      Coil( #Out_Functional_Test.Button_PLC_Functional_Test_25 )
   END_RUNG
   RUNG wire#w1
      Contact( #In_Functional_Test.Electrical_Current_Test_Approved_PLC_Functional_Test_25 )
      Coil( #Out_Functional_Test.Electrical_Current_Test_Approved_PLC_Functional_Test_25 )
   END_RUNG
   RUNG wire#w1
      Contact( #In_Functional_Test.Visual_Test_Approved_PLC_Functional_Test_25 )
      Coil( #Out_Functional_Test.Visual_Test_Approved_PLC_Functional_Test_25 )
   END_RUNG
   RUNG wire#w1
      Move(in := #In_Functional_Test.Electrical_Current_Read_PLC_Functional_Test_25, out1 => #Out_Functional_Test.Electrical_Current_Read_PLC_Functional_Test_25)
   END_RUNG
   RUNG wire#w1
      Contact( #In_Functional_Test.Life_Trigger_PLC_Functional_Test_27 )
      Coil( #Out_Functional_Test.Life_Trigger_PLC_Functional_Test_27 )
   END_RUNG
   RUNG wire#w1
      Contact( #In_Functional_Test.Star_Test_PLC_Functional_Test_27 )
      Coil( #Out_Functional_Test.Star_Test_PLC_Functional_Test_27 )
   END_RUNG
   RUNG wire#w1
      Contact( #In_Functional_Test.Button_PLC_Functional_Test_27 )
      Coil( #Out_Functional_Test.Button_PLC_Functional_Test_27 )
   END_RUNG
   RUNG wire#w1
      Contact( #In_Functional_Test.Electrical_Current_Test_Approved_PLC_Functional_Test_27 )
      Coil( #Out_Functional_Test.Electrical_Current_Test_Approved_PLC_Functional_Test_27 )
   END_RUNG
   RUNG wire#w1
      Contact( #In_Functional_Test.Visual_Test_Approved_PLC_Functional_Test_27 )
      Coil( #Out_Functional_Test.Visual_Test_Approved_PLC_Functional_Test_27 )
   END_RUNG
   RUNG wire#w1
      Move(in := #In_Functional_Test.Electrical_Current_Read_PLC_Functional_Test_27, out1 => #Out_Functional_Test.Electrical_Current_Read_PLC_Functional_Test_27)
   END_RUNG
   RUNG wire#w1
      Contact( #In_Functional_Test.Life_Trigger_PLC_Functional_Test_29 )
      Coil( #Out_Functional_Test.Life_Trigger_PLC_Functional_Test_29 )
   END_RUNG
   RUNG wire#w1
      Contact( #In_Functional_Test.Star_Test_PLC_Functional_Test_29 )
      Coil( #Out_Functional_Test.Star_Test_PLC_Functional_Test_29 )
   END_RUNG
   RUNG wire#w1
      Contact( #In_Functional_Test.Button_PLC_Functional_Test_29 )
      Coil( #Out_Functional_Test.Button_PLC_Functional_Test_29 )
   END_RUNG
   RUNG wire#w1
      Contact( #In_Functional_Test.Electrical_Current_Test_Approved_PLC_Functional_Test_29 )
      Coil( #Out_Functional_Test.Electrical_Current_Test_Approved_PLC_Functional_Test_29 )
   END_RUNG
   RUNG wire#w1
      Contact( #In_Functional_Test.Visual_Test_Approved_PLC_Functional_Test_29 )
      Coil( #Out_Functional_Test.Visual_Test_Approved_PLC_Functional_Test_29 )
   END_RUNG
   RUNG wire#w1
      Move(in := #In_Functional_Test.Electrical_Current_Read_PLC_Functional_Test_29, out1 => #Out_Functional_Test.Electrical_Current_Read_PLC_Functional_Test_29)
   END_RUNG
   // the same network as SCL:
   #_w1 := #Test_Station = 17;
   #Out_Functional_Test.Life_Trigger_PLC_Functional_Test_17 := #_w1 AND #Life_Trigger;
   #Out_Functional_Test.Star_Test_PLC_Functional_Test_17 := #_w1 AND #Star_Test;
   #Out_Functional_Test.Button_PLC_Functional_Test_17 := #_w1 AND #Button_Start_Approve;
   #Out_Functional_Test.Electrical_Current_Test_Approved_PLC_Functional_Test_17 := #_w1 AND #Electrical_Current_Test_Approved;
   #Out_Functional_Test.Visual_Test_Approved_PLC_Functional_Test_17 := #_w1 AND #Visual_Test_Approved;
   #Reset_Functional_Test := #_w1 AND #In_Test_Parameters.Reset_PLC_Functional_Test_17;
   IF #_w1 THEN
       #Out_Functional_Test.Electrical_Current_Read_PLC_Functional_Test_17 := #Electrical_Current_Read;
   END_IF;
   #Out_Functional_Test.Life_Trigger_PLC_Functional_Test_19 := #_w1 AND #In_Functional_Test.Life_Trigger_PLC_Functional_Test_19;
   #Out_Functional_Test.Star_Test_PLC_Functional_Test_19 := #_w1 AND #In_Functional_Test.Star_Test_PLC_Functional_Test_19;
   #Out_Functional_Test.Button_PLC_Functional_Test_19 := #_w1 AND #In_Functional_Test.Button_PLC_Functional_Test_19;
   #Out_Functional_Test.Electrical_Current_Test_Approved_PLC_Functional_Test_19 := #_w1 AND #In_Functional_Test.Electrical_Current_Test_Approved_PLC_Functional_Test_19;
   #Out_Functional_Test.Visual_Test_Approved_PLC_Functional_Test_19 := #_w1 AND #In_Functional_Test.Visual_Test_Approved_PLC_Functional_Test_19;
   IF #_w1 THEN
       #Out_Functional_Test.Electrical_Current_Read_PLC_Functional_Test_19 := #In_Functional_Test.Electrical_Current_Read_PLC_Functional_Test_19;
   END_IF;
   #Out_Functional_Test.Life_Trigger_PLC_Functional_Test_21 := #_w1 AND #In_Functional_Test.Life_Trigger_PLC_Functional_Test_21;
   #Out_Functional_Test.Star_Test_PLC_Functional_Test_21 := #_w1 AND #In_Functional_Test.Star_Test_PLC_Functional_Test_21;
   #Out_Functional_Test.Button_PLC_Functional_Test_21 := #_w1 AND #In_Functional_Test.Button_PLC_Functional_Test_21;
   #Out_Functional_Test.Electrical_Current_Test_Approved_PLC_Functional_Test_21 := #_w1 AND #In_Functional_Test.Electrical_Current_Test_Approved_PLC_Functional_Test_21;
   #Out_Functional_Test.Visual_Test_Approved_PLC_Functional_Test_21 := #_w1 AND #In_Functional_Test.Visual_Test_Approved_PLC_Functional_Test_21;
   IF #_w1 THEN
       #Out_Functional_Test.Electrical_Current_Read_PLC_Functional_Test_21 := #In_Functional_Test.Electrical_Current_Read_PLC_Functional_Test_21;
   END_IF;
   #Out_Functional_Test.Life_Trigger_PLC_Functional_Test_23 := #_w1 AND #In_Functional_Test.Life_Trigger_PLC_Functional_Test_23;
   #Out_Functional_Test.Star_Test_PLC_Functional_Test_23 := #_w1 AND #In_Functional_Test.Star_Test_PLC_Functional_Test_23;
   #Out_Functional_Test.Button_PLC_Functional_Test_23 := #_w1 AND #In_Functional_Test.Button_PLC_Functional_Test_23;
   #Out_Functional_Test.Electrical_Current_Test_Approved_PLC_Functional_Test_23 := #_w1 AND #In_Functional_Test.Electrical_Current_Test_Approved_PLC_Functional_Test_23;
   #Out_Functional_Test.Visual_Test_Approved_PLC_Functional_Test_23 := #_w1 AND #In_Functional_Test.Visual_Test_Approved_PLC_Functional_Test_23;
   IF #_w1 THEN
       #Out_Functional_Test.Electrical_Current_Read_PLC_Functional_Test_23 := #In_Functional_Test.Electrical_Current_Read_PLC_Functional_Test_23;
   END_IF;
   #Out_Functional_Test.Life_Trigger_PLC_Functional_Test_25 := #_w1 AND #In_Functional_Test.Life_Trigger_PLC_Functional_Test_25;
   #Out_Functional_Test.Star_Test_PLC_Functional_Test_25 := #_w1 AND #In_Functional_Test.Star_Test_PLC_Functional_Test_25;
   #Out_Functional_Test.Button_PLC_Functional_Test_25 := #_w1 AND #In_Functional_Test.Button_PLC_Functional_Test_25;
   #Out_Functional_Test.Electrical_Current_Test_Approved_PLC_Functional_Test_25 := #_w1 AND #In_Functional_Test.Electrical_Current_Test_Approved_PLC_Functional_Test_25;
   #Out_Functional_Test.Visual_Test_Approved_PLC_Functional_Test_25 := #_w1 AND #In_Functional_Test.Visual_Test_Approved_PLC_Functional_Test_25;
   IF #_w1 THEN
       #Out_Functional_Test.Electrical_Current_Read_PLC_Functional_Test_25 := #In_Functional_Test.Electrical_Current_Read_PLC_Functional_Test_25;
   END_IF;
   #Out_Functional_Test.Life_Trigger_PLC_Functional_Test_27 := #_w1 AND #In_Functional_Test.Life_Trigger_PLC_Functional_Test_27;
   #Out_Functional_Test.Star_Test_PLC_Functional_Test_27 := #_w1 AND #In_Functional_Test.Star_Test_PLC_Functional_Test_27;
   #Out_Functional_Test.Button_PLC_Functional_Test_27 := #_w1 AND #In_Functional_Test.Button_PLC_Functional_Test_27;
   #Out_Functional_Test.Electrical_Current_Test_Approved_PLC_Functional_Test_27 := #_w1 AND #In_Functional_Test.Electrical_Current_Test_Approved_PLC_Functional_Test_27;
   #Out_Functional_Test.Visual_Test_Approved_PLC_Functional_Test_27 := #_w1 AND #In_Functional_Test.Visual_Test_Approved_PLC_Functional_Test_27;
   IF #_w1 THEN
       #Out_Functional_Test.Electrical_Current_Read_PLC_Functional_Test_27 := #In_Functional_Test.Electrical_Current_Read_PLC_Functional_Test_27;
   END_IF;
   #Out_Functional_Test.Life_Trigger_PLC_Functional_Test_29 := #_w1 AND #In_Functional_Test.Life_Trigger_PLC_Functional_Test_29;
   #Out_Functional_Test.Star_Test_PLC_Functional_Test_29 := #_w1 AND #In_Functional_Test.Star_Test_PLC_Functional_Test_29;
   #Out_Functional_Test.Button_PLC_Functional_Test_29 := #_w1 AND #In_Functional_Test.Button_PLC_Functional_Test_29;
   #Out_Functional_Test.Electrical_Current_Test_Approved_PLC_Functional_Test_29 := #_w1 AND #In_Functional_Test.Electrical_Current_Test_Approved_PLC_Functional_Test_29;
   #Out_Functional_Test.Visual_Test_Approved_PLC_Functional_Test_29 := #_w1 AND #In_Functional_Test.Visual_Test_Approved_PLC_Functional_Test_29;
   IF #_w1 THEN
       #Out_Functional_Test.Electrical_Current_Read_PLC_Functional_Test_29 := #In_Functional_Test.Electrical_Current_Read_PLC_Functional_Test_29;
   END_IF;
END_REGION

REGION Network 11: Functional Test Station 19
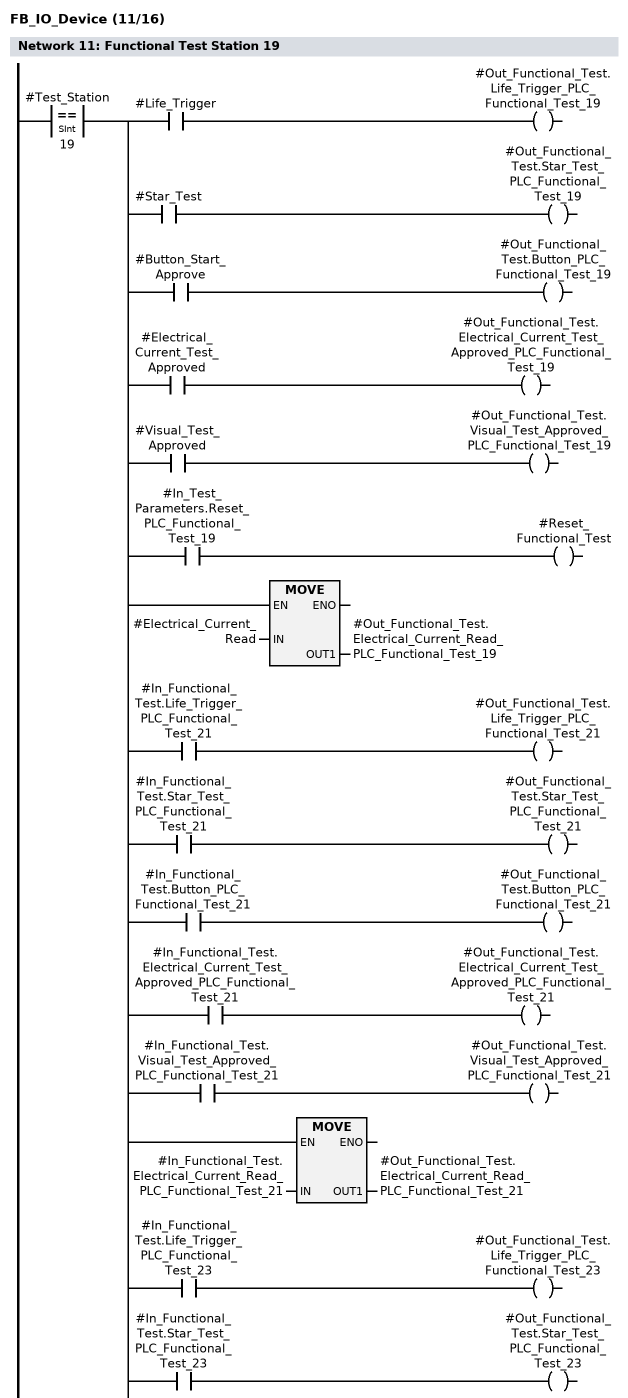
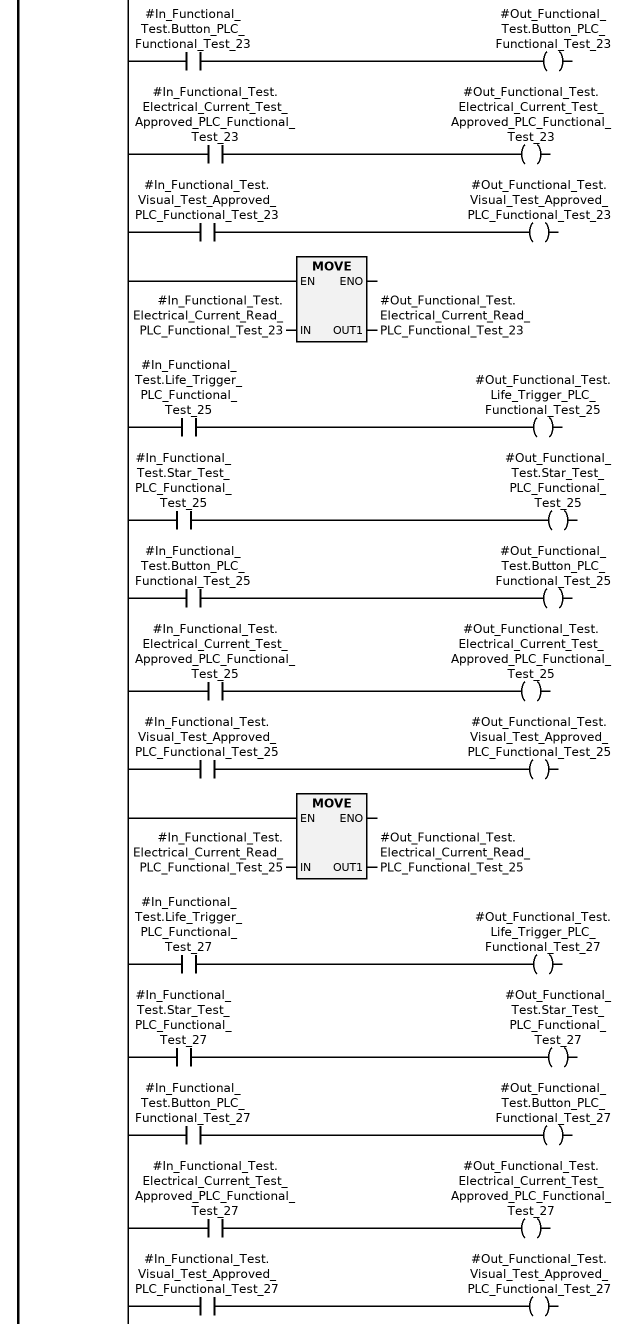
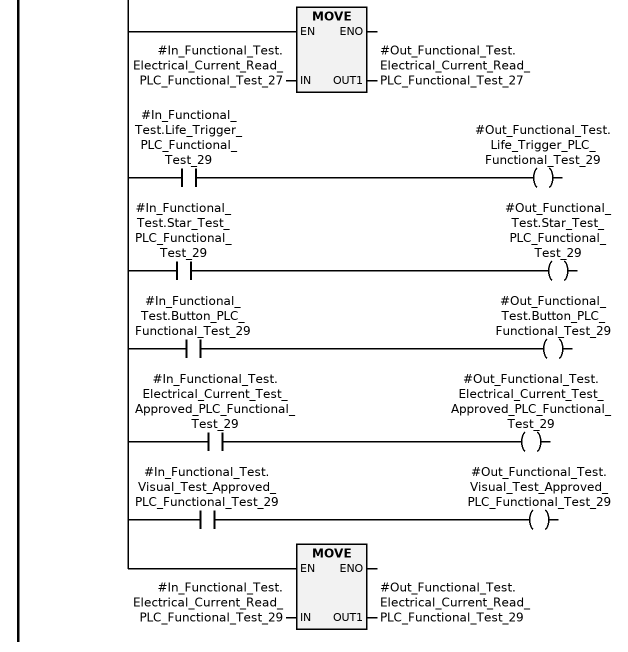
   RUNG wire#powerrail
      { S7_Templates := "SrcType := SInt" } EQ_Contact(in1 := #Test_Station, in2 := 19)
      wire#w1
      Contact( #Life_Trigger )
      Coil( #Out_Functional_Test.Life_Trigger_PLC_Functional_Test_19 )
   END_RUNG
   RUNG wire#w1
      Contact( #Star_Test )
      Coil( #Out_Functional_Test.Star_Test_PLC_Functional_Test_19 )
   END_RUNG
   RUNG wire#w1
      Contact( #Button_Start_Approve )
      Coil( #Out_Functional_Test.Button_PLC_Functional_Test_19 )
   END_RUNG
   RUNG wire#w1
      Contact( #Electrical_Current_Test_Approved )
      Coil( #Out_Functional_Test.Electrical_Current_Test_Approved_PLC_Functional_Test_19 )
   END_RUNG
   RUNG wire#w1
      Contact( #Visual_Test_Approved )
      Coil( #Out_Functional_Test.Visual_Test_Approved_PLC_Functional_Test_19 )
   END_RUNG
   RUNG wire#w1
      Contact( #In_Test_Parameters.Reset_PLC_Functional_Test_19 )
      Coil( #Reset_Functional_Test )
   END_RUNG
   RUNG wire#w1
      Move(in := #Electrical_Current_Read, out1 => #Out_Functional_Test.Electrical_Current_Read_PLC_Functional_Test_19)
   END_RUNG
   RUNG wire#w1
      Contact( #In_Functional_Test.Life_Trigger_PLC_Functional_Test_21 )
      Coil( #Out_Functional_Test.Life_Trigger_PLC_Functional_Test_21 )
   END_RUNG
   RUNG wire#w1
      Contact( #In_Functional_Test.Star_Test_PLC_Functional_Test_21 )
      Coil( #Out_Functional_Test.Star_Test_PLC_Functional_Test_21 )
   END_RUNG
   RUNG wire#w1
      Contact( #In_Functional_Test.Button_PLC_Functional_Test_21 )
      Coil( #Out_Functional_Test.Button_PLC_Functional_Test_21 )
   END_RUNG
   RUNG wire#w1
      Contact( #In_Functional_Test.Electrical_Current_Test_Approved_PLC_Functional_Test_21 )
      Coil( #Out_Functional_Test.Electrical_Current_Test_Approved_PLC_Functional_Test_21 )
   END_RUNG
   RUNG wire#w1
      Contact( #In_Functional_Test.Visual_Test_Approved_PLC_Functional_Test_21 )
      Coil( #Out_Functional_Test.Visual_Test_Approved_PLC_Functional_Test_21 )
   END_RUNG
   RUNG wire#w1
      Move(in := #In_Functional_Test.Electrical_Current_Read_PLC_Functional_Test_21, out1 => #Out_Functional_Test.Electrical_Current_Read_PLC_Functional_Test_21)
   END_RUNG
   RUNG wire#w1
      Contact( #In_Functional_Test.Life_Trigger_PLC_Functional_Test_23 )
      Coil( #Out_Functional_Test.Life_Trigger_PLC_Functional_Test_23 )
   END_RUNG
   RUNG wire#w1
      Contact( #In_Functional_Test.Star_Test_PLC_Functional_Test_23 )
      Coil( #Out_Functional_Test.Star_Test_PLC_Functional_Test_23 )
   END_RUNG
   RUNG wire#w1
      Contact( #In_Functional_Test.Button_PLC_Functional_Test_23 )
      Coil( #Out_Functional_Test.Button_PLC_Functional_Test_23 )
   END_RUNG
   RUNG wire#w1
      Contact( #In_Functional_Test.Electrical_Current_Test_Approved_PLC_Functional_Test_23 )
      Coil( #Out_Functional_Test.Electrical_Current_Test_Approved_PLC_Functional_Test_23 )
   END_RUNG
   RUNG wire#w1
      Contact( #In_Functional_Test.Visual_Test_Approved_PLC_Functional_Test_23 )
      Coil( #Out_Functional_Test.Visual_Test_Approved_PLC_Functional_Test_23 )
   END_RUNG
   RUNG wire#w1
      Move(in := #In_Functional_Test.Electrical_Current_Read_PLC_Functional_Test_23, out1 => #Out_Functional_Test.Electrical_Current_Read_PLC_Functional_Test_23)
   END_RUNG
   RUNG wire#w1
      Contact( #In_Functional_Test.Life_Trigger_PLC_Functional_Test_25 )
      Coil( #Out_Functional_Test.Life_Trigger_PLC_Functional_Test_25 )
   END_RUNG
   RUNG wire#w1
      Contact( #In_Functional_Test.Star_Test_PLC_Functional_Test_25 )
      Coil( #Out_Functional_Test.Star_Test_PLC_Functional_Test_25 )
   END_RUNG
   RUNG wire#w1
      Contact( #In_Functional_Test.Button_PLC_Functional_Test_25 )
      Coil( #Out_Functional_Test.Button_PLC_Functional_Test_25 )
   END_RUNG
   RUNG wire#w1
      Contact( #In_Functional_Test.Electrical_Current_Test_Approved_PLC_Functional_Test_25 )
      Coil( #Out_Functional_Test.Electrical_Current_Test_Approved_PLC_Functional_Test_25 )
   END_RUNG
   RUNG wire#w1
      Contact( #In_Functional_Test.Visual_Test_Approved_PLC_Functional_Test_25 )
      Coil( #Out_Functional_Test.Visual_Test_Approved_PLC_Functional_Test_25 )
   END_RUNG
   RUNG wire#w1
      Move(in := #In_Functional_Test.Electrical_Current_Read_PLC_Functional_Test_25, out1 => #Out_Functional_Test.Electrical_Current_Read_PLC_Functional_Test_25)
   END_RUNG
   RUNG wire#w1
      Contact( #In_Functional_Test.Life_Trigger_PLC_Functional_Test_27 )
      Coil( #Out_Functional_Test.Life_Trigger_PLC_Functional_Test_27 )
   END_RUNG
   RUNG wire#w1
      Contact( #In_Functional_Test.Star_Test_PLC_Functional_Test_27 )
      Coil( #Out_Functional_Test.Star_Test_PLC_Functional_Test_27 )
   END_RUNG
   RUNG wire#w1
      Contact( #In_Functional_Test.Button_PLC_Functional_Test_27 )
      Coil( #Out_Functional_Test.Button_PLC_Functional_Test_27 )
   END_RUNG
   RUNG wire#w1
      Contact( #In_Functional_Test.Electrical_Current_Test_Approved_PLC_Functional_Test_27 )
      Coil( #Out_Functional_Test.Electrical_Current_Test_Approved_PLC_Functional_Test_27 )
   END_RUNG
   RUNG wire#w1
      Contact( #In_Functional_Test.Visual_Test_Approved_PLC_Functional_Test_27 )
      Coil( #Out_Functional_Test.Visual_Test_Approved_PLC_Functional_Test_27 )
   END_RUNG
   RUNG wire#w1
      Move(in := #In_Functional_Test.Electrical_Current_Read_PLC_Functional_Test_27, out1 => #Out_Functional_Test.Electrical_Current_Read_PLC_Functional_Test_27)
   END_RUNG
   RUNG wire#w1
      Contact( #In_Functional_Test.Life_Trigger_PLC_Functional_Test_29 )
      Coil( #Out_Functional_Test.Life_Trigger_PLC_Functional_Test_29 )
   END_RUNG
   RUNG wire#w1
      Contact( #In_Functional_Test.Star_Test_PLC_Functional_Test_29 )
      Coil( #Out_Functional_Test.Star_Test_PLC_Functional_Test_29 )
   END_RUNG
   RUNG wire#w1
      Contact( #In_Functional_Test.Button_PLC_Functional_Test_29 )
      Coil( #Out_Functional_Test.Button_PLC_Functional_Test_29 )
   END_RUNG
   RUNG wire#w1
      Contact( #In_Functional_Test.Electrical_Current_Test_Approved_PLC_Functional_Test_29 )
      Coil( #Out_Functional_Test.Electrical_Current_Test_Approved_PLC_Functional_Test_29 )
   END_RUNG
   RUNG wire#w1
      Contact( #In_Functional_Test.Visual_Test_Approved_PLC_Functional_Test_29 )
      Coil( #Out_Functional_Test.Visual_Test_Approved_PLC_Functional_Test_29 )
   END_RUNG
   RUNG wire#w1
      Move(in := #In_Functional_Test.Electrical_Current_Read_PLC_Functional_Test_29, out1 => #Out_Functional_Test.Electrical_Current_Read_PLC_Functional_Test_29)
   END_RUNG
   // the same network as SCL:
   #_w1 := #Test_Station = 19;
   #Out_Functional_Test.Life_Trigger_PLC_Functional_Test_19 := #_w1 AND #Life_Trigger;
   #Out_Functional_Test.Star_Test_PLC_Functional_Test_19 := #_w1 AND #Star_Test;
   #Out_Functional_Test.Button_PLC_Functional_Test_19 := #_w1 AND #Button_Start_Approve;
   #Out_Functional_Test.Electrical_Current_Test_Approved_PLC_Functional_Test_19 := #_w1 AND #Electrical_Current_Test_Approved;
   #Out_Functional_Test.Visual_Test_Approved_PLC_Functional_Test_19 := #_w1 AND #Visual_Test_Approved;
   #Reset_Functional_Test := #_w1 AND #In_Test_Parameters.Reset_PLC_Functional_Test_19;
   IF #_w1 THEN
       #Out_Functional_Test.Electrical_Current_Read_PLC_Functional_Test_19 := #Electrical_Current_Read;
   END_IF;
   #Out_Functional_Test.Life_Trigger_PLC_Functional_Test_21 := #_w1 AND #In_Functional_Test.Life_Trigger_PLC_Functional_Test_21;
   #Out_Functional_Test.Star_Test_PLC_Functional_Test_21 := #_w1 AND #In_Functional_Test.Star_Test_PLC_Functional_Test_21;
   #Out_Functional_Test.Button_PLC_Functional_Test_21 := #_w1 AND #In_Functional_Test.Button_PLC_Functional_Test_21;
   #Out_Functional_Test.Electrical_Current_Test_Approved_PLC_Functional_Test_21 := #_w1 AND #In_Functional_Test.Electrical_Current_Test_Approved_PLC_Functional_Test_21;
   #Out_Functional_Test.Visual_Test_Approved_PLC_Functional_Test_21 := #_w1 AND #In_Functional_Test.Visual_Test_Approved_PLC_Functional_Test_21;
   IF #_w1 THEN
       #Out_Functional_Test.Electrical_Current_Read_PLC_Functional_Test_21 := #In_Functional_Test.Electrical_Current_Read_PLC_Functional_Test_21;
   END_IF;
   #Out_Functional_Test.Life_Trigger_PLC_Functional_Test_23 := #_w1 AND #In_Functional_Test.Life_Trigger_PLC_Functional_Test_23;
   #Out_Functional_Test.Star_Test_PLC_Functional_Test_23 := #_w1 AND #In_Functional_Test.Star_Test_PLC_Functional_Test_23;
   #Out_Functional_Test.Button_PLC_Functional_Test_23 := #_w1 AND #In_Functional_Test.Button_PLC_Functional_Test_23;
   #Out_Functional_Test.Electrical_Current_Test_Approved_PLC_Functional_Test_23 := #_w1 AND #In_Functional_Test.Electrical_Current_Test_Approved_PLC_Functional_Test_23;
   #Out_Functional_Test.Visual_Test_Approved_PLC_Functional_Test_23 := #_w1 AND #In_Functional_Test.Visual_Test_Approved_PLC_Functional_Test_23;
   IF #_w1 THEN
       #Out_Functional_Test.Electrical_Current_Read_PLC_Functional_Test_23 := #In_Functional_Test.Electrical_Current_Read_PLC_Functional_Test_23;
   END_IF;
   #Out_Functional_Test.Life_Trigger_PLC_Functional_Test_25 := #_w1 AND #In_Functional_Test.Life_Trigger_PLC_Functional_Test_25;
   #Out_Functional_Test.Star_Test_PLC_Functional_Test_25 := #_w1 AND #In_Functional_Test.Star_Test_PLC_Functional_Test_25;
   #Out_Functional_Test.Button_PLC_Functional_Test_25 := #_w1 AND #In_Functional_Test.Button_PLC_Functional_Test_25;
   #Out_Functional_Test.Electrical_Current_Test_Approved_PLC_Functional_Test_25 := #_w1 AND #In_Functional_Test.Electrical_Current_Test_Approved_PLC_Functional_Test_25;
   #Out_Functional_Test.Visual_Test_Approved_PLC_Functional_Test_25 := #_w1 AND #In_Functional_Test.Visual_Test_Approved_PLC_Functional_Test_25;
   IF #_w1 THEN
       #Out_Functional_Test.Electrical_Current_Read_PLC_Functional_Test_25 := #In_Functional_Test.Electrical_Current_Read_PLC_Functional_Test_25;
   END_IF;
   #Out_Functional_Test.Life_Trigger_PLC_Functional_Test_27 := #_w1 AND #In_Functional_Test.Life_Trigger_PLC_Functional_Test_27;
   #Out_Functional_Test.Star_Test_PLC_Functional_Test_27 := #_w1 AND #In_Functional_Test.Star_Test_PLC_Functional_Test_27;
   #Out_Functional_Test.Button_PLC_Functional_Test_27 := #_w1 AND #In_Functional_Test.Button_PLC_Functional_Test_27;
   #Out_Functional_Test.Electrical_Current_Test_Approved_PLC_Functional_Test_27 := #_w1 AND #In_Functional_Test.Electrical_Current_Test_Approved_PLC_Functional_Test_27;
   #Out_Functional_Test.Visual_Test_Approved_PLC_Functional_Test_27 := #_w1 AND #In_Functional_Test.Visual_Test_Approved_PLC_Functional_Test_27;
   IF #_w1 THEN
       #Out_Functional_Test.Electrical_Current_Read_PLC_Functional_Test_27 := #In_Functional_Test.Electrical_Current_Read_PLC_Functional_Test_27;
   END_IF;
   #Out_Functional_Test.Life_Trigger_PLC_Functional_Test_29 := #_w1 AND #In_Functional_Test.Life_Trigger_PLC_Functional_Test_29;
   #Out_Functional_Test.Star_Test_PLC_Functional_Test_29 := #_w1 AND #In_Functional_Test.Star_Test_PLC_Functional_Test_29;
   #Out_Functional_Test.Button_PLC_Functional_Test_29 := #_w1 AND #In_Functional_Test.Button_PLC_Functional_Test_29;
   #Out_Functional_Test.Electrical_Current_Test_Approved_PLC_Functional_Test_29 := #_w1 AND #In_Functional_Test.Electrical_Current_Test_Approved_PLC_Functional_Test_29;
   #Out_Functional_Test.Visual_Test_Approved_PLC_Functional_Test_29 := #_w1 AND #In_Functional_Test.Visual_Test_Approved_PLC_Functional_Test_29;
   IF #_w1 THEN
       #Out_Functional_Test.Electrical_Current_Read_PLC_Functional_Test_29 := #In_Functional_Test.Electrical_Current_Read_PLC_Functional_Test_29;
   END_IF;
END_REGION

REGION Network 12: Functional Test Station 21
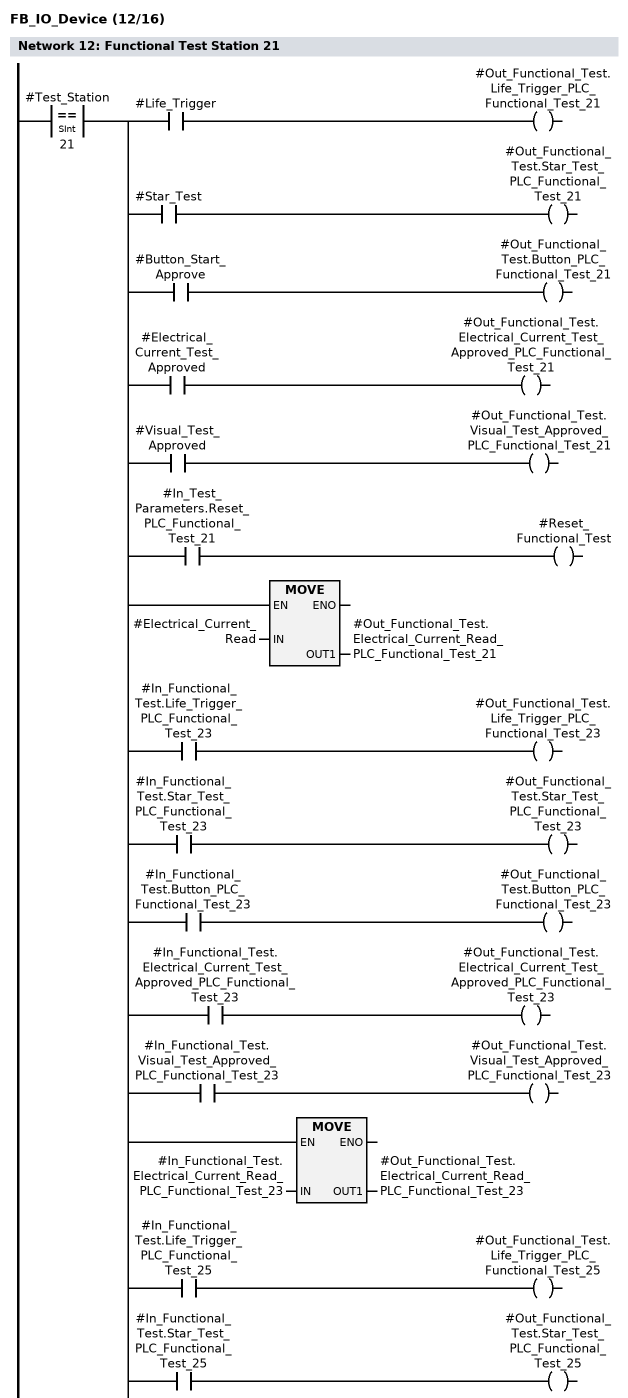
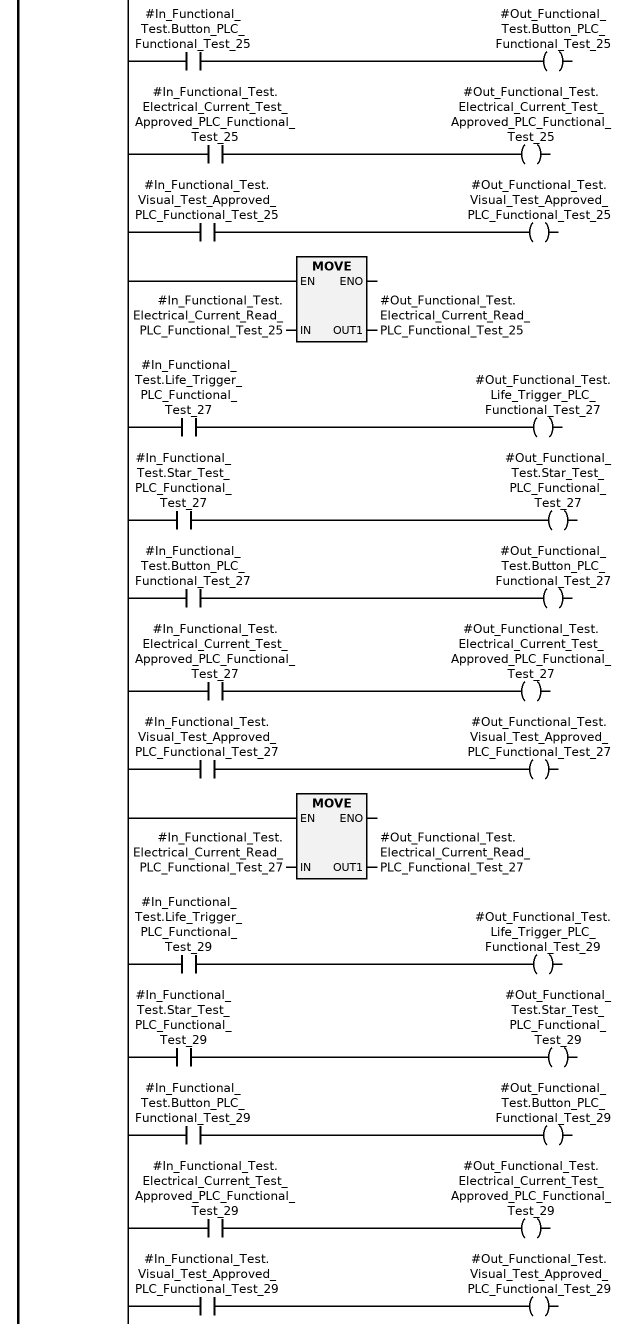
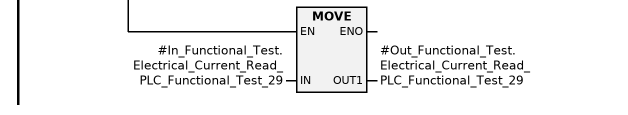
   RUNG wire#powerrail
      { S7_Templates := "SrcType := SInt" } EQ_Contact(in1 := #Test_Station, in2 := 21)
      wire#w1
      Contact( #Life_Trigger )
      Coil( #Out_Functional_Test.Life_Trigger_PLC_Functional_Test_21 )
   END_RUNG
   RUNG wire#w1
      Contact( #Star_Test )
      Coil( #Out_Functional_Test.Star_Test_PLC_Functional_Test_21 )
   END_RUNG
   RUNG wire#w1
      Contact( #Button_Start_Approve )
      Coil( #Out_Functional_Test.Button_PLC_Functional_Test_21 )
   END_RUNG
   RUNG wire#w1
      Contact( #Electrical_Current_Test_Approved )
      Coil( #Out_Functional_Test.Electrical_Current_Test_Approved_PLC_Functional_Test_21 )
   END_RUNG
   RUNG wire#w1
      Contact( #Visual_Test_Approved )
      Coil( #Out_Functional_Test.Visual_Test_Approved_PLC_Functional_Test_21 )
   END_RUNG
   RUNG wire#w1
      Contact( #In_Test_Parameters.Reset_PLC_Functional_Test_21 )
      Coil( #Reset_Functional_Test )
   END_RUNG
   RUNG wire#w1
      Move(in := #Electrical_Current_Read, out1 => #Out_Functional_Test.Electrical_Current_Read_PLC_Functional_Test_21)
   END_RUNG
   RUNG wire#w1
      Contact( #In_Functional_Test.Life_Trigger_PLC_Functional_Test_23 )
      Coil( #Out_Functional_Test.Life_Trigger_PLC_Functional_Test_23 )
   END_RUNG
   RUNG wire#w1
      Contact( #In_Functional_Test.Star_Test_PLC_Functional_Test_23 )
      Coil( #Out_Functional_Test.Star_Test_PLC_Functional_Test_23 )
   END_RUNG
   RUNG wire#w1
      Contact( #In_Functional_Test.Button_PLC_Functional_Test_23 )
      Coil( #Out_Functional_Test.Button_PLC_Functional_Test_23 )
   END_RUNG
   RUNG wire#w1
      Contact( #In_Functional_Test.Electrical_Current_Test_Approved_PLC_Functional_Test_23 )
      Coil( #Out_Functional_Test.Electrical_Current_Test_Approved_PLC_Functional_Test_23 )
   END_RUNG
   RUNG wire#w1
      Contact( #In_Functional_Test.Visual_Test_Approved_PLC_Functional_Test_23 )
      Coil( #Out_Functional_Test.Visual_Test_Approved_PLC_Functional_Test_23 )
   END_RUNG
   RUNG wire#w1
      Move(in := #In_Functional_Test.Electrical_Current_Read_PLC_Functional_Test_23, out1 => #Out_Functional_Test.Electrical_Current_Read_PLC_Functional_Test_23)
   END_RUNG
   RUNG wire#w1
      Contact( #In_Functional_Test.Life_Trigger_PLC_Functional_Test_25 )
      Coil( #Out_Functional_Test.Life_Trigger_PLC_Functional_Test_25 )
   END_RUNG
   RUNG wire#w1
      Contact( #In_Functional_Test.Star_Test_PLC_Functional_Test_25 )
      Coil( #Out_Functional_Test.Star_Test_PLC_Functional_Test_25 )
   END_RUNG
   RUNG wire#w1
      Contact( #In_Functional_Test.Button_PLC_Functional_Test_25 )
      Coil( #Out_Functional_Test.Button_PLC_Functional_Test_25 )
   END_RUNG
   RUNG wire#w1
      Contact( #In_Functional_Test.Electrical_Current_Test_Approved_PLC_Functional_Test_25 )
      Coil( #Out_Functional_Test.Electrical_Current_Test_Approved_PLC_Functional_Test_25 )
   END_RUNG
   RUNG wire#w1
      Contact( #In_Functional_Test.Visual_Test_Approved_PLC_Functional_Test_25 )
      Coil( #Out_Functional_Test.Visual_Test_Approved_PLC_Functional_Test_25 )
   END_RUNG
   RUNG wire#w1
      Move(in := #In_Functional_Test.Electrical_Current_Read_PLC_Functional_Test_25, out1 => #Out_Functional_Test.Electrical_Current_Read_PLC_Functional_Test_25)
   END_RUNG
   RUNG wire#w1
      Contact( #In_Functional_Test.Life_Trigger_PLC_Functional_Test_27 )
      Coil( #Out_Functional_Test.Life_Trigger_PLC_Functional_Test_27 )
   END_RUNG
   RUNG wire#w1
      Contact( #In_Functional_Test.Star_Test_PLC_Functional_Test_27 )
      Coil( #Out_Functional_Test.Star_Test_PLC_Functional_Test_27 )
   END_RUNG
   RUNG wire#w1
      Contact( #In_Functional_Test.Button_PLC_Functional_Test_27 )
      Coil( #Out_Functional_Test.Button_PLC_Functional_Test_27 )
   END_RUNG
   RUNG wire#w1
      Contact( #In_Functional_Test.Electrical_Current_Test_Approved_PLC_Functional_Test_27 )
      Coil( #Out_Functional_Test.Electrical_Current_Test_Approved_PLC_Functional_Test_27 )
   END_RUNG
   RUNG wire#w1
      Contact( #In_Functional_Test.Visual_Test_Approved_PLC_Functional_Test_27 )
      Coil( #Out_Functional_Test.Visual_Test_Approved_PLC_Functional_Test_27 )
   END_RUNG
   RUNG wire#w1
      Move(in := #In_Functional_Test.Electrical_Current_Read_PLC_Functional_Test_27, out1 => #Out_Functional_Test.Electrical_Current_Read_PLC_Functional_Test_27)
   END_RUNG
   RUNG wire#w1
      Contact( #In_Functional_Test.Life_Trigger_PLC_Functional_Test_29 )
      Coil( #Out_Functional_Test.Life_Trigger_PLC_Functional_Test_29 )
   END_RUNG
   RUNG wire#w1
      Contact( #In_Functional_Test.Star_Test_PLC_Functional_Test_29 )
      Coil( #Out_Functional_Test.Star_Test_PLC_Functional_Test_29 )
   END_RUNG
   RUNG wire#w1
      Contact( #In_Functional_Test.Button_PLC_Functional_Test_29 )
      Coil( #Out_Functional_Test.Button_PLC_Functional_Test_29 )
   END_RUNG
   RUNG wire#w1
      Contact( #In_Functional_Test.Electrical_Current_Test_Approved_PLC_Functional_Test_29 )
      Coil( #Out_Functional_Test.Electrical_Current_Test_Approved_PLC_Functional_Test_29 )
   END_RUNG
   RUNG wire#w1
      Contact( #In_Functional_Test.Visual_Test_Approved_PLC_Functional_Test_29 )
      Coil( #Out_Functional_Test.Visual_Test_Approved_PLC_Functional_Test_29 )
   END_RUNG
   RUNG wire#w1
      Move(in := #In_Functional_Test.Electrical_Current_Read_PLC_Functional_Test_29, out1 => #Out_Functional_Test.Electrical_Current_Read_PLC_Functional_Test_29)
   END_RUNG
   // the same network as SCL:
   #_w1 := #Test_Station = 21;
   #Out_Functional_Test.Life_Trigger_PLC_Functional_Test_21 := #_w1 AND #Life_Trigger;
   #Out_Functional_Test.Star_Test_PLC_Functional_Test_21 := #_w1 AND #Star_Test;
   #Out_Functional_Test.Button_PLC_Functional_Test_21 := #_w1 AND #Button_Start_Approve;
   #Out_Functional_Test.Electrical_Current_Test_Approved_PLC_Functional_Test_21 := #_w1 AND #Electrical_Current_Test_Approved;
   #Out_Functional_Test.Visual_Test_Approved_PLC_Functional_Test_21 := #_w1 AND #Visual_Test_Approved;
   #Reset_Functional_Test := #_w1 AND #In_Test_Parameters.Reset_PLC_Functional_Test_21;
   IF #_w1 THEN
       #Out_Functional_Test.Electrical_Current_Read_PLC_Functional_Test_21 := #Electrical_Current_Read;
   END_IF;
   #Out_Functional_Test.Life_Trigger_PLC_Functional_Test_23 := #_w1 AND #In_Functional_Test.Life_Trigger_PLC_Functional_Test_23;
   #Out_Functional_Test.Star_Test_PLC_Functional_Test_23 := #_w1 AND #In_Functional_Test.Star_Test_PLC_Functional_Test_23;
   #Out_Functional_Test.Button_PLC_Functional_Test_23 := #_w1 AND #In_Functional_Test.Button_PLC_Functional_Test_23;
   #Out_Functional_Test.Electrical_Current_Test_Approved_PLC_Functional_Test_23 := #_w1 AND #In_Functional_Test.Electrical_Current_Test_Approved_PLC_Functional_Test_23;
   #Out_Functional_Test.Visual_Test_Approved_PLC_Functional_Test_23 := #_w1 AND #In_Functional_Test.Visual_Test_Approved_PLC_Functional_Test_23;
   IF #_w1 THEN
       #Out_Functional_Test.Electrical_Current_Read_PLC_Functional_Test_23 := #In_Functional_Test.Electrical_Current_Read_PLC_Functional_Test_23;
   END_IF;
   #Out_Functional_Test.Life_Trigger_PLC_Functional_Test_25 := #_w1 AND #In_Functional_Test.Life_Trigger_PLC_Functional_Test_25;
   #Out_Functional_Test.Star_Test_PLC_Functional_Test_25 := #_w1 AND #In_Functional_Test.Star_Test_PLC_Functional_Test_25;
   #Out_Functional_Test.Button_PLC_Functional_Test_25 := #_w1 AND #In_Functional_Test.Button_PLC_Functional_Test_25;
   #Out_Functional_Test.Electrical_Current_Test_Approved_PLC_Functional_Test_25 := #_w1 AND #In_Functional_Test.Electrical_Current_Test_Approved_PLC_Functional_Test_25;
   #Out_Functional_Test.Visual_Test_Approved_PLC_Functional_Test_25 := #_w1 AND #In_Functional_Test.Visual_Test_Approved_PLC_Functional_Test_25;
   IF #_w1 THEN
       #Out_Functional_Test.Electrical_Current_Read_PLC_Functional_Test_25 := #In_Functional_Test.Electrical_Current_Read_PLC_Functional_Test_25;
   END_IF;
   #Out_Functional_Test.Life_Trigger_PLC_Functional_Test_27 := #_w1 AND #In_Functional_Test.Life_Trigger_PLC_Functional_Test_27;
   #Out_Functional_Test.Star_Test_PLC_Functional_Test_27 := #_w1 AND #In_Functional_Test.Star_Test_PLC_Functional_Test_27;
   #Out_Functional_Test.Button_PLC_Functional_Test_27 := #_w1 AND #In_Functional_Test.Button_PLC_Functional_Test_27;
   #Out_Functional_Test.Electrical_Current_Test_Approved_PLC_Functional_Test_27 := #_w1 AND #In_Functional_Test.Electrical_Current_Test_Approved_PLC_Functional_Test_27;
   #Out_Functional_Test.Visual_Test_Approved_PLC_Functional_Test_27 := #_w1 AND #In_Functional_Test.Visual_Test_Approved_PLC_Functional_Test_27;
   IF #_w1 THEN
       #Out_Functional_Test.Electrical_Current_Read_PLC_Functional_Test_27 := #In_Functional_Test.Electrical_Current_Read_PLC_Functional_Test_27;
   END_IF;
   #Out_Functional_Test.Life_Trigger_PLC_Functional_Test_29 := #_w1 AND #In_Functional_Test.Life_Trigger_PLC_Functional_Test_29;
   #Out_Functional_Test.Star_Test_PLC_Functional_Test_29 := #_w1 AND #In_Functional_Test.Star_Test_PLC_Functional_Test_29;
   #Out_Functional_Test.Button_PLC_Functional_Test_29 := #_w1 AND #In_Functional_Test.Button_PLC_Functional_Test_29;
   #Out_Functional_Test.Electrical_Current_Test_Approved_PLC_Functional_Test_29 := #_w1 AND #In_Functional_Test.Electrical_Current_Test_Approved_PLC_Functional_Test_29;
   #Out_Functional_Test.Visual_Test_Approved_PLC_Functional_Test_29 := #_w1 AND #In_Functional_Test.Visual_Test_Approved_PLC_Functional_Test_29;
   IF #_w1 THEN
       #Out_Functional_Test.Electrical_Current_Read_PLC_Functional_Test_29 := #In_Functional_Test.Electrical_Current_Read_PLC_Functional_Test_29;
   END_IF;
END_REGION

REGION Network 13: Functional Test Station 23
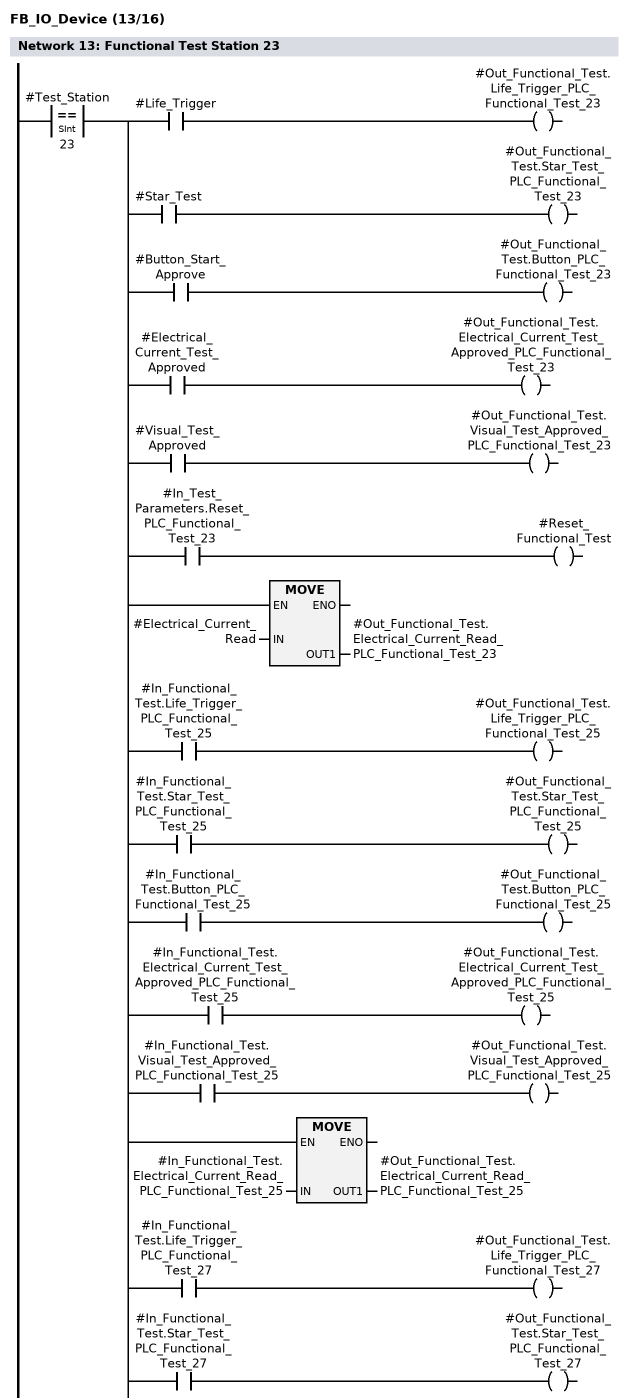
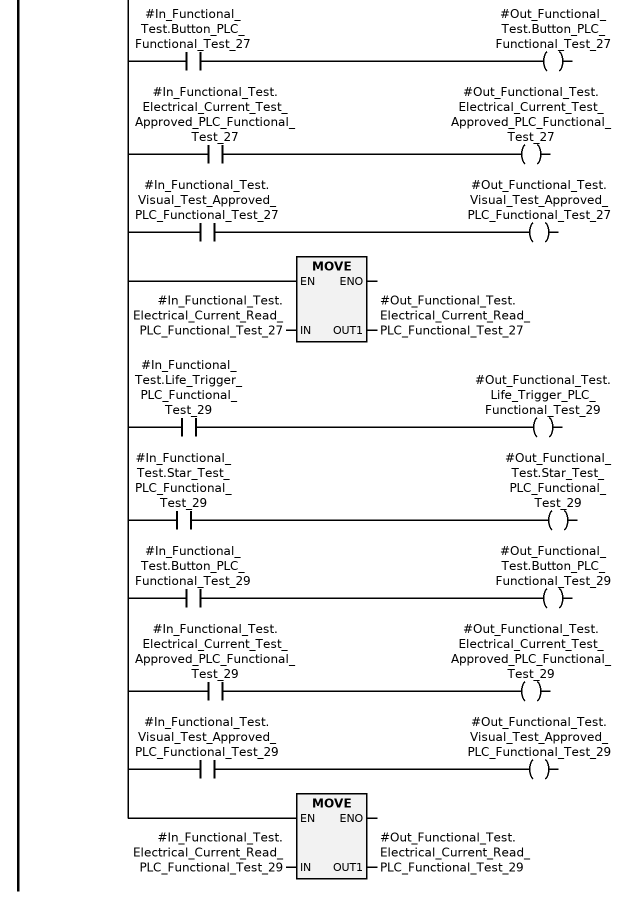
   RUNG wire#powerrail
      { S7_Templates := "SrcType := SInt" } EQ_Contact(in1 := #Test_Station, in2 := 23)
      wire#w1
      Contact( #Life_Trigger )
      Coil( #Out_Functional_Test.Life_Trigger_PLC_Functional_Test_23 )
   END_RUNG
   RUNG wire#w1
      Contact( #Star_Test )
      Coil( #Out_Functional_Test.Star_Test_PLC_Functional_Test_23 )
   END_RUNG
   RUNG wire#w1
      Contact( #Button_Start_Approve )
      Coil( #Out_Functional_Test.Button_PLC_Functional_Test_23 )
   END_RUNG
   RUNG wire#w1
      Contact( #Electrical_Current_Test_Approved )
      Coil( #Out_Functional_Test.Electrical_Current_Test_Approved_PLC_Functional_Test_23 )
   END_RUNG
   RUNG wire#w1
      Contact( #Visual_Test_Approved )
      Coil( #Out_Functional_Test.Visual_Test_Approved_PLC_Functional_Test_23 )
   END_RUNG
   RUNG wire#w1
      Contact( #In_Test_Parameters.Reset_PLC_Functional_Test_23 )
      Coil( #Reset_Functional_Test )
   END_RUNG
   RUNG wire#w1
      Move(in := #Electrical_Current_Read, out1 => #Out_Functional_Test.Electrical_Current_Read_PLC_Functional_Test_23)
   END_RUNG
   RUNG wire#w1
      Contact( #In_Functional_Test.Life_Trigger_PLC_Functional_Test_25 )
      Coil( #Out_Functional_Test.Life_Trigger_PLC_Functional_Test_25 )
   END_RUNG
   RUNG wire#w1
      Contact( #In_Functional_Test.Star_Test_PLC_Functional_Test_25 )
      Coil( #Out_Functional_Test.Star_Test_PLC_Functional_Test_25 )
   END_RUNG
   RUNG wire#w1
      Contact( #In_Functional_Test.Button_PLC_Functional_Test_25 )
      Coil( #Out_Functional_Test.Button_PLC_Functional_Test_25 )
   END_RUNG
   RUNG wire#w1
      Contact( #In_Functional_Test.Electrical_Current_Test_Approved_PLC_Functional_Test_25 )
      Coil( #Out_Functional_Test.Electrical_Current_Test_Approved_PLC_Functional_Test_25 )
   END_RUNG
   RUNG wire#w1
      Contact( #In_Functional_Test.Visual_Test_Approved_PLC_Functional_Test_25 )
      Coil( #Out_Functional_Test.Visual_Test_Approved_PLC_Functional_Test_25 )
   END_RUNG
   RUNG wire#w1
      Move(in := #In_Functional_Test.Electrical_Current_Read_PLC_Functional_Test_25, out1 => #Out_Functional_Test.Electrical_Current_Read_PLC_Functional_Test_25)
   END_RUNG
   RUNG wire#w1
      Contact( #In_Functional_Test.Life_Trigger_PLC_Functional_Test_27 )
      Coil( #Out_Functional_Test.Life_Trigger_PLC_Functional_Test_27 )
   END_RUNG
   RUNG wire#w1
      Contact( #In_Functional_Test.Star_Test_PLC_Functional_Test_27 )
      Coil( #Out_Functional_Test.Star_Test_PLC_Functional_Test_27 )
   END_RUNG
   RUNG wire#w1
      Contact( #In_Functional_Test.Button_PLC_Functional_Test_27 )
      Coil( #Out_Functional_Test.Button_PLC_Functional_Test_27 )
   END_RUNG
   RUNG wire#w1
      Contact( #In_Functional_Test.Electrical_Current_Test_Approved_PLC_Functional_Test_27 )
      Coil( #Out_Functional_Test.Electrical_Current_Test_Approved_PLC_Functional_Test_27 )
   END_RUNG
   RUNG wire#w1
      Contact( #In_Functional_Test.Visual_Test_Approved_PLC_Functional_Test_27 )
      Coil( #Out_Functional_Test.Visual_Test_Approved_PLC_Functional_Test_27 )
   END_RUNG
   RUNG wire#w1
      Move(in := #In_Functional_Test.Electrical_Current_Read_PLC_Functional_Test_27, out1 => #Out_Functional_Test.Electrical_Current_Read_PLC_Functional_Test_27)
   END_RUNG
   RUNG wire#w1
      Contact( #In_Functional_Test.Life_Trigger_PLC_Functional_Test_29 )
      Coil( #Out_Functional_Test.Life_Trigger_PLC_Functional_Test_29 )
   END_RUNG
   RUNG wire#w1
      Contact( #In_Functional_Test.Star_Test_PLC_Functional_Test_29 )
      Coil( #Out_Functional_Test.Star_Test_PLC_Functional_Test_29 )
   END_RUNG
   RUNG wire#w1
      Contact( #In_Functional_Test.Button_PLC_Functional_Test_29 )
      Coil( #Out_Functional_Test.Button_PLC_Functional_Test_29 )
   END_RUNG
   RUNG wire#w1
      Contact( #In_Functional_Test.Electrical_Current_Test_Approved_PLC_Functional_Test_29 )
      Coil( #Out_Functional_Test.Electrical_Current_Test_Approved_PLC_Functional_Test_29 )
   END_RUNG
   RUNG wire#w1
      Contact( #In_Functional_Test.Visual_Test_Approved_PLC_Functional_Test_29 )
      Coil( #Out_Functional_Test.Visual_Test_Approved_PLC_Functional_Test_29 )
   END_RUNG
   RUNG wire#w1
      Move(in := #In_Functional_Test.Electrical_Current_Read_PLC_Functional_Test_29, out1 => #Out_Functional_Test.Electrical_Current_Read_PLC_Functional_Test_29)
   END_RUNG
   // the same network as SCL:
   #_w1 := #Test_Station = 23;
   #Out_Functional_Test.Life_Trigger_PLC_Functional_Test_23 := #_w1 AND #Life_Trigger;
   #Out_Functional_Test.Star_Test_PLC_Functional_Test_23 := #_w1 AND #Star_Test;
   #Out_Functional_Test.Button_PLC_Functional_Test_23 := #_w1 AND #Button_Start_Approve;
   #Out_Functional_Test.Electrical_Current_Test_Approved_PLC_Functional_Test_23 := #_w1 AND #Electrical_Current_Test_Approved;
   #Out_Functional_Test.Visual_Test_Approved_PLC_Functional_Test_23 := #_w1 AND #Visual_Test_Approved;
   #Reset_Functional_Test := #_w1 AND #In_Test_Parameters.Reset_PLC_Functional_Test_23;
   IF #_w1 THEN
       #Out_Functional_Test.Electrical_Current_Read_PLC_Functional_Test_23 := #Electrical_Current_Read;
   END_IF;
   #Out_Functional_Test.Life_Trigger_PLC_Functional_Test_25 := #_w1 AND #In_Functional_Test.Life_Trigger_PLC_Functional_Test_25;
   #Out_Functional_Test.Star_Test_PLC_Functional_Test_25 := #_w1 AND #In_Functional_Test.Star_Test_PLC_Functional_Test_25;
   #Out_Functional_Test.Button_PLC_Functional_Test_25 := #_w1 AND #In_Functional_Test.Button_PLC_Functional_Test_25;
   #Out_Functional_Test.Electrical_Current_Test_Approved_PLC_Functional_Test_25 := #_w1 AND #In_Functional_Test.Electrical_Current_Test_Approved_PLC_Functional_Test_25;
   #Out_Functional_Test.Visual_Test_Approved_PLC_Functional_Test_25 := #_w1 AND #In_Functional_Test.Visual_Test_Approved_PLC_Functional_Test_25;
   IF #_w1 THEN
       #Out_Functional_Test.Electrical_Current_Read_PLC_Functional_Test_25 := #In_Functional_Test.Electrical_Current_Read_PLC_Functional_Test_25;
   END_IF;
   #Out_Functional_Test.Life_Trigger_PLC_Functional_Test_27 := #_w1 AND #In_Functional_Test.Life_Trigger_PLC_Functional_Test_27;
   #Out_Functional_Test.Star_Test_PLC_Functional_Test_27 := #_w1 AND #In_Functional_Test.Star_Test_PLC_Functional_Test_27;
   #Out_Functional_Test.Button_PLC_Functional_Test_27 := #_w1 AND #In_Functional_Test.Button_PLC_Functional_Test_27;
   #Out_Functional_Test.Electrical_Current_Test_Approved_PLC_Functional_Test_27 := #_w1 AND #In_Functional_Test.Electrical_Current_Test_Approved_PLC_Functional_Test_27;
   #Out_Functional_Test.Visual_Test_Approved_PLC_Functional_Test_27 := #_w1 AND #In_Functional_Test.Visual_Test_Approved_PLC_Functional_Test_27;
   IF #_w1 THEN
       #Out_Functional_Test.Electrical_Current_Read_PLC_Functional_Test_27 := #In_Functional_Test.Electrical_Current_Read_PLC_Functional_Test_27;
   END_IF;
   #Out_Functional_Test.Life_Trigger_PLC_Functional_Test_29 := #_w1 AND #In_Functional_Test.Life_Trigger_PLC_Functional_Test_29;
   #Out_Functional_Test.Star_Test_PLC_Functional_Test_29 := #_w1 AND #In_Functional_Test.Star_Test_PLC_Functional_Test_29;
   #Out_Functional_Test.Button_PLC_Functional_Test_29 := #_w1 AND #In_Functional_Test.Button_PLC_Functional_Test_29;
   #Out_Functional_Test.Electrical_Current_Test_Approved_PLC_Functional_Test_29 := #_w1 AND #In_Functional_Test.Electrical_Current_Test_Approved_PLC_Functional_Test_29;
   #Out_Functional_Test.Visual_Test_Approved_PLC_Functional_Test_29 := #_w1 AND #In_Functional_Test.Visual_Test_Approved_PLC_Functional_Test_29;
   IF #_w1 THEN
       #Out_Functional_Test.Electrical_Current_Read_PLC_Functional_Test_29 := #In_Functional_Test.Electrical_Current_Read_PLC_Functional_Test_29;
   END_IF;
END_REGION

REGION Network 14: Functional Test Station 25
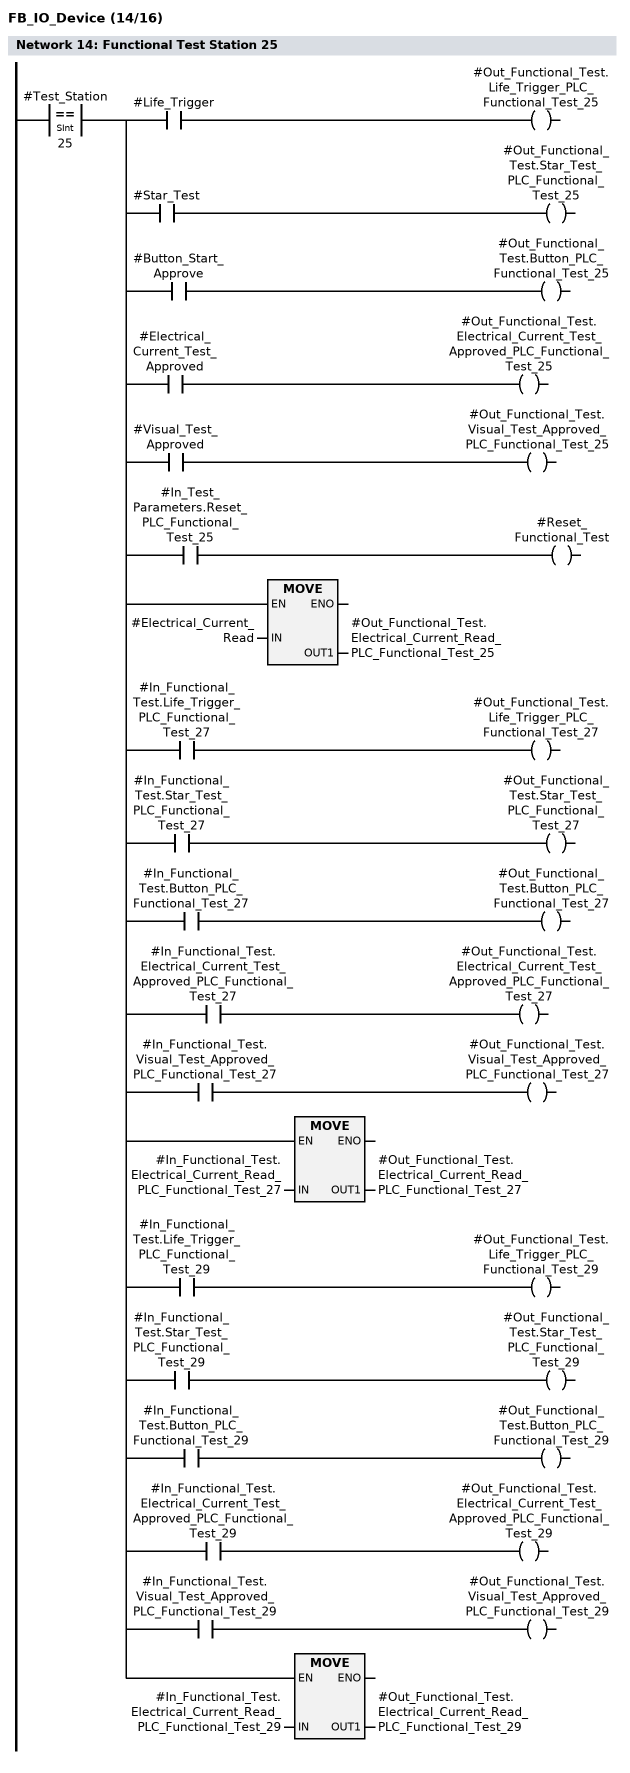
   RUNG wire#powerrail
      { S7_Templates := "SrcType := SInt" } EQ_Contact(in1 := #Test_Station, in2 := 25)
      wire#w1
      Contact( #Life_Trigger )
      Coil( #Out_Functional_Test.Life_Trigger_PLC_Functional_Test_25 )
   END_RUNG
   RUNG wire#w1
      Contact( #Star_Test )
      Coil( #Out_Functional_Test.Star_Test_PLC_Functional_Test_25 )
   END_RUNG
   RUNG wire#w1
      Contact( #Button_Start_Approve )
      Coil( #Out_Functional_Test.Button_PLC_Functional_Test_25 )
   END_RUNG
   RUNG wire#w1
      Contact( #Electrical_Current_Test_Approved )
      Coil( #Out_Functional_Test.Electrical_Current_Test_Approved_PLC_Functional_Test_25 )
   END_RUNG
   RUNG wire#w1
      Contact( #Visual_Test_Approved )
      Coil( #Out_Functional_Test.Visual_Test_Approved_PLC_Functional_Test_25 )
   END_RUNG
   RUNG wire#w1
      Contact( #In_Test_Parameters.Reset_PLC_Functional_Test_25 )
      Coil( #Reset_Functional_Test )
   END_RUNG
   RUNG wire#w1
      Move(in := #Electrical_Current_Read, out1 => #Out_Functional_Test.Electrical_Current_Read_PLC_Functional_Test_25)
   END_RUNG
   RUNG wire#w1
      Contact( #In_Functional_Test.Life_Trigger_PLC_Functional_Test_27 )
      Coil( #Out_Functional_Test.Life_Trigger_PLC_Functional_Test_27 )
   END_RUNG
   RUNG wire#w1
      Contact( #In_Functional_Test.Star_Test_PLC_Functional_Test_27 )
      Coil( #Out_Functional_Test.Star_Test_PLC_Functional_Test_27 )
   END_RUNG
   RUNG wire#w1
      Contact( #In_Functional_Test.Button_PLC_Functional_Test_27 )
      Coil( #Out_Functional_Test.Button_PLC_Functional_Test_27 )
   END_RUNG
   RUNG wire#w1
      Contact( #In_Functional_Test.Electrical_Current_Test_Approved_PLC_Functional_Test_27 )
      Coil( #Out_Functional_Test.Electrical_Current_Test_Approved_PLC_Functional_Test_27 )
   END_RUNG
   RUNG wire#w1
      Contact( #In_Functional_Test.Visual_Test_Approved_PLC_Functional_Test_27 )
      Coil( #Out_Functional_Test.Visual_Test_Approved_PLC_Functional_Test_27 )
   END_RUNG
   RUNG wire#w1
      Move(in := #In_Functional_Test.Electrical_Current_Read_PLC_Functional_Test_27, out1 => #Out_Functional_Test.Electrical_Current_Read_PLC_Functional_Test_27)
   END_RUNG
   RUNG wire#w1
      Contact( #In_Functional_Test.Life_Trigger_PLC_Functional_Test_29 )
      Coil( #Out_Functional_Test.Life_Trigger_PLC_Functional_Test_29 )
   END_RUNG
   RUNG wire#w1
      Contact( #In_Functional_Test.Star_Test_PLC_Functional_Test_29 )
      Coil( #Out_Functional_Test.Star_Test_PLC_Functional_Test_29 )
   END_RUNG
   RUNG wire#w1
      Contact( #In_Functional_Test.Button_PLC_Functional_Test_29 )
      Coil( #Out_Functional_Test.Button_PLC_Functional_Test_29 )
   END_RUNG
   RUNG wire#w1
      Contact( #In_Functional_Test.Electrical_Current_Test_Approved_PLC_Functional_Test_29 )
      Coil( #Out_Functional_Test.Electrical_Current_Test_Approved_PLC_Functional_Test_29 )
   END_RUNG
   RUNG wire#w1
      Contact( #In_Functional_Test.Visual_Test_Approved_PLC_Functional_Test_29 )
      Coil( #Out_Functional_Test.Visual_Test_Approved_PLC_Functional_Test_29 )
   END_RUNG
   RUNG wire#w1
      Move(in := #In_Functional_Test.Electrical_Current_Read_PLC_Functional_Test_29, out1 => #Out_Functional_Test.Electrical_Current_Read_PLC_Functional_Test_29)
   END_RUNG
   // the same network as SCL:
   #_w1 := #Test_Station = 25;
   #Out_Functional_Test.Life_Trigger_PLC_Functional_Test_25 := #_w1 AND #Life_Trigger;
   #Out_Functional_Test.Star_Test_PLC_Functional_Test_25 := #_w1 AND #Star_Test;
   #Out_Functional_Test.Button_PLC_Functional_Test_25 := #_w1 AND #Button_Start_Approve;
   #Out_Functional_Test.Electrical_Current_Test_Approved_PLC_Functional_Test_25 := #_w1 AND #Electrical_Current_Test_Approved;
   #Out_Functional_Test.Visual_Test_Approved_PLC_Functional_Test_25 := #_w1 AND #Visual_Test_Approved;
   #Reset_Functional_Test := #_w1 AND #In_Test_Parameters.Reset_PLC_Functional_Test_25;
   IF #_w1 THEN
       #Out_Functional_Test.Electrical_Current_Read_PLC_Functional_Test_25 := #Electrical_Current_Read;
   END_IF;
   #Out_Functional_Test.Life_Trigger_PLC_Functional_Test_27 := #_w1 AND #In_Functional_Test.Life_Trigger_PLC_Functional_Test_27;
   #Out_Functional_Test.Star_Test_PLC_Functional_Test_27 := #_w1 AND #In_Functional_Test.Star_Test_PLC_Functional_Test_27;
   #Out_Functional_Test.Button_PLC_Functional_Test_27 := #_w1 AND #In_Functional_Test.Button_PLC_Functional_Test_27;
   #Out_Functional_Test.Electrical_Current_Test_Approved_PLC_Functional_Test_27 := #_w1 AND #In_Functional_Test.Electrical_Current_Test_Approved_PLC_Functional_Test_27;
   #Out_Functional_Test.Visual_Test_Approved_PLC_Functional_Test_27 := #_w1 AND #In_Functional_Test.Visual_Test_Approved_PLC_Functional_Test_27;
   IF #_w1 THEN
       #Out_Functional_Test.Electrical_Current_Read_PLC_Functional_Test_27 := #In_Functional_Test.Electrical_Current_Read_PLC_Functional_Test_27;
   END_IF;
   #Out_Functional_Test.Life_Trigger_PLC_Functional_Test_29 := #_w1 AND #In_Functional_Test.Life_Trigger_PLC_Functional_Test_29;
   #Out_Functional_Test.Star_Test_PLC_Functional_Test_29 := #_w1 AND #In_Functional_Test.Star_Test_PLC_Functional_Test_29;
   #Out_Functional_Test.Button_PLC_Functional_Test_29 := #_w1 AND #In_Functional_Test.Button_PLC_Functional_Test_29;
   #Out_Functional_Test.Electrical_Current_Test_Approved_PLC_Functional_Test_29 := #_w1 AND #In_Functional_Test.Electrical_Current_Test_Approved_PLC_Functional_Test_29;
   #Out_Functional_Test.Visual_Test_Approved_PLC_Functional_Test_29 := #_w1 AND #In_Functional_Test.Visual_Test_Approved_PLC_Functional_Test_29;
   IF #_w1 THEN
       #Out_Functional_Test.Electrical_Current_Read_PLC_Functional_Test_29 := #In_Functional_Test.Electrical_Current_Read_PLC_Functional_Test_29;
   END_IF;
END_REGION

REGION Network 15: Functional Test Station 27
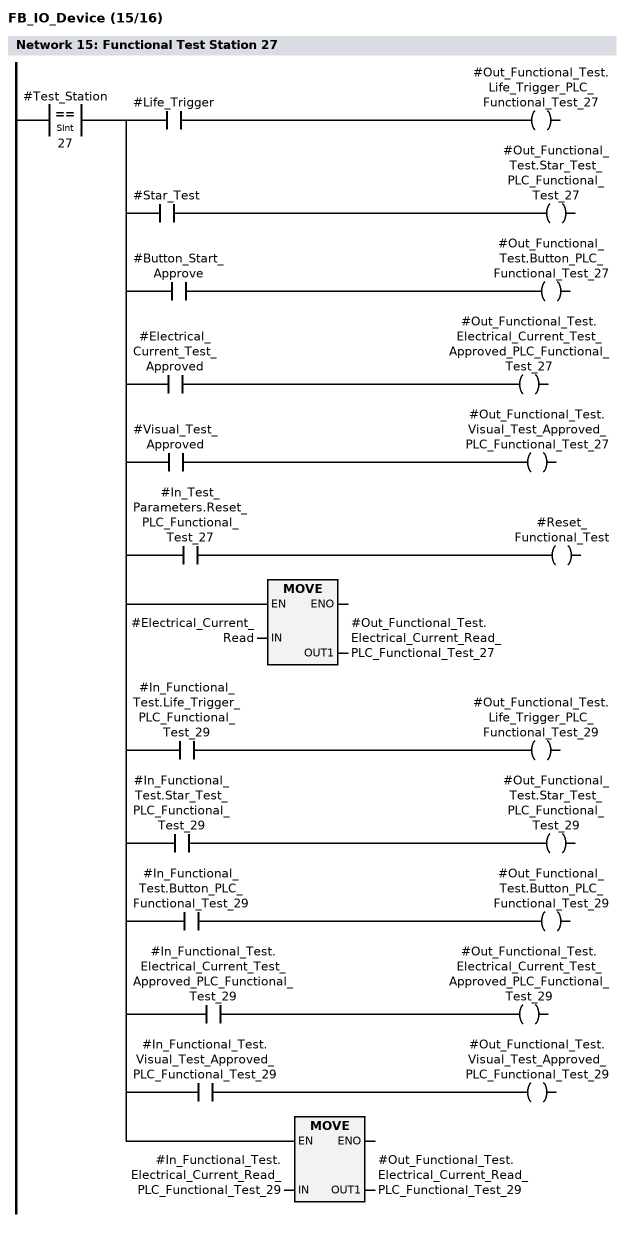
   RUNG wire#powerrail
      { S7_Templates := "SrcType := SInt" } EQ_Contact(in1 := #Test_Station, in2 := 27)
      wire#w1
      Contact( #Life_Trigger )
      Coil( #Out_Functional_Test.Life_Trigger_PLC_Functional_Test_27 )
   END_RUNG
   RUNG wire#w1
      Contact( #Star_Test )
      Coil( #Out_Functional_Test.Star_Test_PLC_Functional_Test_27 )
   END_RUNG
   RUNG wire#w1
      Contact( #Button_Start_Approve )
      Coil( #Out_Functional_Test.Button_PLC_Functional_Test_27 )
   END_RUNG
   RUNG wire#w1
      Contact( #Electrical_Current_Test_Approved )
      Coil( #Out_Functional_Test.Electrical_Current_Test_Approved_PLC_Functional_Test_27 )
   END_RUNG
   RUNG wire#w1
      Contact( #Visual_Test_Approved )
      Coil( #Out_Functional_Test.Visual_Test_Approved_PLC_Functional_Test_27 )
   END_RUNG
   RUNG wire#w1
      Contact( #In_Test_Parameters.Reset_PLC_Functional_Test_27 )
      Coil( #Reset_Functional_Test )
   END_RUNG
   RUNG wire#w1
      Move(in := #Electrical_Current_Read, out1 => #Out_Functional_Test.Electrical_Current_Read_PLC_Functional_Test_27)
   END_RUNG
   RUNG wire#w1
      Contact( #In_Functional_Test.Life_Trigger_PLC_Functional_Test_29 )
      Coil( #Out_Functional_Test.Life_Trigger_PLC_Functional_Test_29 )
   END_RUNG
   RUNG wire#w1
      Contact( #In_Functional_Test.Star_Test_PLC_Functional_Test_29 )
      Coil( #Out_Functional_Test.Star_Test_PLC_Functional_Test_29 )
   END_RUNG
   RUNG wire#w1
      Contact( #In_Functional_Test.Button_PLC_Functional_Test_29 )
      Coil( #Out_Functional_Test.Button_PLC_Functional_Test_29 )
   END_RUNG
   RUNG wire#w1
      Contact( #In_Functional_Test.Electrical_Current_Test_Approved_PLC_Functional_Test_29 )
      Coil( #Out_Functional_Test.Electrical_Current_Test_Approved_PLC_Functional_Test_29 )
   END_RUNG
   RUNG wire#w1
      Contact( #In_Functional_Test.Visual_Test_Approved_PLC_Functional_Test_29 )
      Coil( #Out_Functional_Test.Visual_Test_Approved_PLC_Functional_Test_29 )
   END_RUNG
   RUNG wire#w1
      Move(in := #In_Functional_Test.Electrical_Current_Read_PLC_Functional_Test_29, out1 => #Out_Functional_Test.Electrical_Current_Read_PLC_Functional_Test_29)
   END_RUNG
   // the same network as SCL:
   #_w1 := #Test_Station = 27;
   #Out_Functional_Test.Life_Trigger_PLC_Functional_Test_27 := #_w1 AND #Life_Trigger;
   #Out_Functional_Test.Star_Test_PLC_Functional_Test_27 := #_w1 AND #Star_Test;
   #Out_Functional_Test.Button_PLC_Functional_Test_27 := #_w1 AND #Button_Start_Approve;
   #Out_Functional_Test.Electrical_Current_Test_Approved_PLC_Functional_Test_27 := #_w1 AND #Electrical_Current_Test_Approved;
   #Out_Functional_Test.Visual_Test_Approved_PLC_Functional_Test_27 := #_w1 AND #Visual_Test_Approved;
   #Reset_Functional_Test := #_w1 AND #In_Test_Parameters.Reset_PLC_Functional_Test_27;
   IF #_w1 THEN
       #Out_Functional_Test.Electrical_Current_Read_PLC_Functional_Test_27 := #Electrical_Current_Read;
   END_IF;
   #Out_Functional_Test.Life_Trigger_PLC_Functional_Test_29 := #_w1 AND #In_Functional_Test.Life_Trigger_PLC_Functional_Test_29;
   #Out_Functional_Test.Star_Test_PLC_Functional_Test_29 := #_w1 AND #In_Functional_Test.Star_Test_PLC_Functional_Test_29;
   #Out_Functional_Test.Button_PLC_Functional_Test_29 := #_w1 AND #In_Functional_Test.Button_PLC_Functional_Test_29;
   #Out_Functional_Test.Electrical_Current_Test_Approved_PLC_Functional_Test_29 := #_w1 AND #In_Functional_Test.Electrical_Current_Test_Approved_PLC_Functional_Test_29;
   #Out_Functional_Test.Visual_Test_Approved_PLC_Functional_Test_29 := #_w1 AND #In_Functional_Test.Visual_Test_Approved_PLC_Functional_Test_29;
   IF #_w1 THEN
       #Out_Functional_Test.Electrical_Current_Read_PLC_Functional_Test_29 := #In_Functional_Test.Electrical_Current_Read_PLC_Functional_Test_29;
   END_IF;
END_REGION

REGION Network 16: Functional Test Station 29
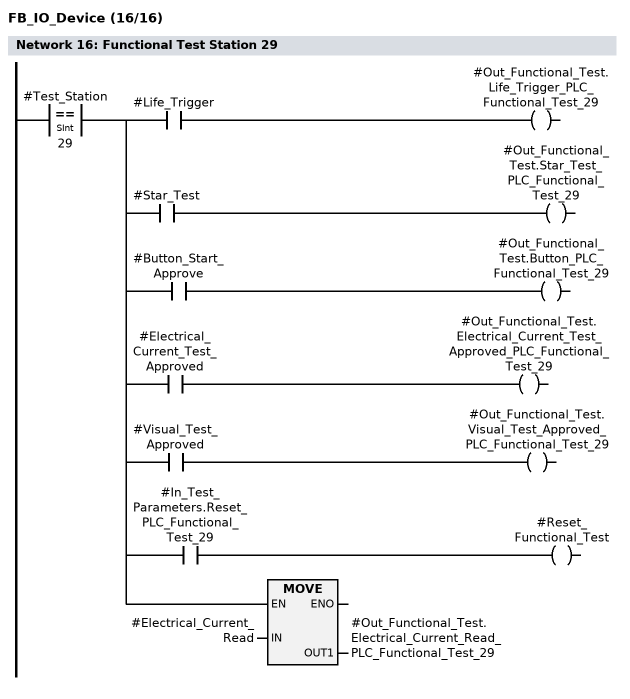
   RUNG wire#powerrail
      { S7_Templates := "SrcType := SInt" } EQ_Contact(in1 := #Test_Station, in2 := 29)
      wire#w1
      Contact( #Life_Trigger )
      Coil( #Out_Functional_Test.Life_Trigger_PLC_Functional_Test_29 )
   END_RUNG
   RUNG wire#w1
      Contact( #Star_Test )
      Coil( #Out_Functional_Test.Star_Test_PLC_Functional_Test_29 )
   END_RUNG
   RUNG wire#w1
      Contact( #Button_Start_Approve )
      Coil( #Out_Functional_Test.Button_PLC_Functional_Test_29 )
   END_RUNG
   RUNG wire#w1
      Contact( #Electrical_Current_Test_Approved )
      Coil( #Out_Functional_Test.Electrical_Current_Test_Approved_PLC_Functional_Test_29 )
   END_RUNG
   RUNG wire#w1
      Contact( #Visual_Test_Approved )
      Coil( #Out_Functional_Test.Visual_Test_Approved_PLC_Functional_Test_29 )
   END_RUNG
   RUNG wire#w1
      Contact( #In_Test_Parameters.Reset_PLC_Functional_Test_29 )
      Coil( #Reset_Functional_Test )
   END_RUNG
   RUNG wire#w1
      Move(in := #Electrical_Current_Read, out1 => #Out_Functional_Test.Electrical_Current_Read_PLC_Functional_Test_29)
   END_RUNG
   // the same network as SCL:
   #_w1 := #Test_Station = 29;
   #Out_Functional_Test.Life_Trigger_PLC_Functional_Test_29 := #_w1 AND #Life_Trigger;
   #Out_Functional_Test.Star_Test_PLC_Functional_Test_29 := #_w1 AND #Star_Test;
   #Out_Functional_Test.Button_PLC_Functional_Test_29 := #_w1 AND #Button_Start_Approve;
   #Out_Functional_Test.Electrical_Current_Test_Approved_PLC_Functional_Test_29 := #_w1 AND #Electrical_Current_Test_Approved;
   #Out_Functional_Test.Visual_Test_Approved_PLC_Functional_Test_29 := #_w1 AND #Visual_Test_Approved;
   #Reset_Functional_Test := #_w1 AND #In_Test_Parameters.Reset_PLC_Functional_Test_29;
   IF #_w1 THEN
       #Out_Functional_Test.Electrical_Current_Read_PLC_Functional_Test_29 := #Electrical_Current_Read;
   END_IF;
END_REGION
END_FUNCTION_BLOCK

FUNCTION_BLOCK "FB_Start_Test"   // FB5, LAD
{ S7_Optimized_Access := 'TRUE' }
// stored: MemoryReserve 100, SetENOAutomatically false
   VAR_INPUT
      Button_Start_Approve : Bool;
      Electrical_Current_Test_Approved : Bool;
      Visual_Test_Approved_PLC : Bool;
      Reset_Funcional_Test : Bool;
   END_VAR
   VAR_OUTPUT
      Start_Functional_Test : Bool;
      Blink_Button_Light : Bool;
      Turn_On_Button_Light : Bool;
      Light_Fail_Test : Bool;
      Light_Approve_Test : Bool;
   END_VAR
   VAR
      Aux_Trigger_0 : Bool;
   END_VAR
   VAR_TEMP   // added for the SCL form of the ladder/FBD networks
      _w1 : Bool;
      _w2 : Bool;
   END_VAR
BEGIN

REGION Network 1: Set Start Functional Test, Blink the Button Light, Turn on Red Light (Fail Test)
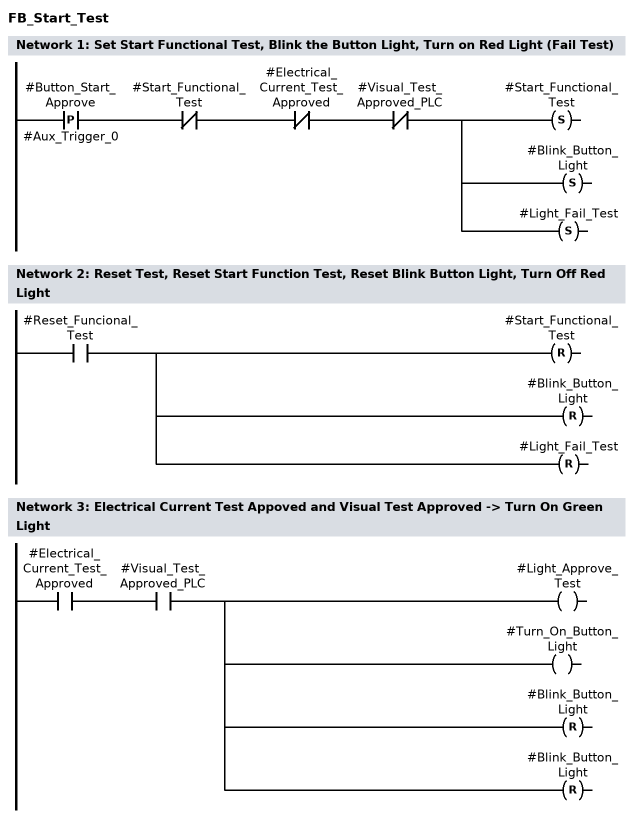
   RUNG wire#powerrail
      P_Contact(operand := #Button_Start_Approve, bit := #Aux_Trigger_0)
      I_Contact( #Start_Functional_Test )
      I_Contact( #Electrical_Current_Test_Approved )
      I_Contact( #Visual_Test_Approved_PLC )
      wire#w1
      S_Coil( #Start_Functional_Test )
   END_RUNG
   RUNG wire#w1
      S_Coil( #Blink_Button_Light )
   END_RUNG
   RUNG wire#w1
      S_Coil( #Light_Fail_Test )
   END_RUNG
   // the same network as SCL:
   #_w1 := #Button_Start_Approve AND NOT #Aux_Trigger_0;   // rising edge of #Button_Start_Approve
   #Aux_Trigger_0 := #Button_Start_Approve;
   #_w2 := #_w1 AND NOT #Start_Functional_Test AND NOT #Electrical_Current_Test_Approved AND NOT #Visual_Test_Approved_PLC;
   IF #_w2 THEN
       #Start_Functional_Test := TRUE;
       #Blink_Button_Light := TRUE;
       #Light_Fail_Test := TRUE;
   END_IF;
END_REGION

REGION Network 2: Reset Test, Reset Start Function Test, Reset Blink Button Light, Turn Off Red Light
   RUNG wire#powerrail
      Contact( #Reset_Funcional_Test )
      wire#w1
      R_Coil( #Start_Functional_Test )
   END_RUNG
   RUNG wire#w1
      R_Coil( #Blink_Button_Light )
   END_RUNG
   RUNG wire#w1
      R_Coil( #Light_Fail_Test )
   END_RUNG
   // the same network as SCL:
   IF #Reset_Funcional_Test THEN
       #Start_Functional_Test := FALSE;
       #Blink_Button_Light := FALSE;
       #Light_Fail_Test := FALSE;
   END_IF;
END_REGION

REGION Network 3: Electrical Current Test Appoved and Visual Test Approved -> Turn On Green Light
   RUNG wire#powerrail
      Contact( #Electrical_Current_Test_Approved )
      Contact( #Visual_Test_Approved_PLC )
      wire#w1
      Coil( #Light_Approve_Test )
   END_RUNG
   RUNG wire#w1
      Coil( #Turn_On_Button_Light )
   END_RUNG
   RUNG wire#w1
      R_Coil( #Blink_Button_Light )
   END_RUNG
   RUNG wire#w1
      R_Coil( #Blink_Button_Light )
   END_RUNG
   // the same network as SCL:
   #Light_Approve_Test := #Electrical_Current_Test_Approved AND #Visual_Test_Approved_PLC;
   #Turn_On_Button_Light := #Light_Approve_Test;
   IF #Light_Approve_Test THEN
       #Blink_Button_Light := FALSE;
       #Blink_Button_Light := FALSE;
   END_IF;
END_REGION
END_FUNCTION_BLOCK

FUNCTION_BLOCK "FB_Visual_Test"   // FB7, LAD
{ S7_Optimized_Access := 'TRUE' }
// stored: MemoryReserve 100, SetENOAutomatically false
   VAR_INPUT
      Star_Functional_Test : Bool;
      Reset_Functional_Test : Bool;
      Button_Start_Approve : Bool;
      In_Test_Parameters : "IO_Device_Test_Parameters";
   END_VAR
   VAR_OUTPUT
      Visual_Test_Approved_PLC : Bool;
   END_VAR
   VAR
      Aux_Trigger : Bool;
      Timer_Delay_Start_Visual_Test { S7_SetPoint := 'True'} : TON_TIME;
      Timer_Delay_Reset { S7_SetPoint := 'True'} : TON_TIME;
   END_VAR
   VAR_TEMP   // added for the SCL form of the ladder/FBD networks
      _w1 : Bool;
   END_VAR
BEGIN

REGION Network 1
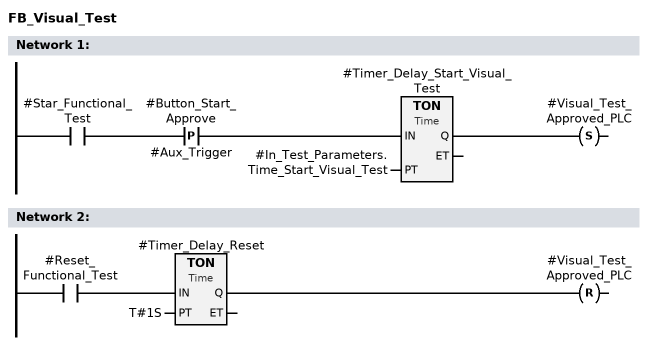
   RUNG wire#powerrail
      Contact( #Star_Functional_Test )
      P_Contact(operand := #Button_Start_Approve, bit := #Aux_Trigger)
      { S7_Templates := "time_type := Time" } #Timer_Delay_Start_Visual_Test.TON(pt := #In_Test_Parameters.Time_Start_Visual_Test, et =>)
      S_Coil( #Visual_Test_Approved_PLC )
   END_RUNG
   // the same network as SCL:
   #_w1 := #Star_Functional_Test AND #Button_Start_Approve AND NOT #Aux_Trigger;   // rising edge of #Button_Start_Approve
   #Aux_Trigger := #Button_Start_Approve;
   #Timer_Delay_Start_Visual_Test(IN := #_w1, PT := #In_Test_Parameters.Time_Start_Visual_Test);   // TON
   IF #Timer_Delay_Start_Visual_Test.Q THEN #Visual_Test_Approved_PLC := TRUE; END_IF;
END_REGION

REGION Network 2
   RUNG wire#powerrail
      Contact( #Reset_Functional_Test )
      { S7_Templates := "time_type := Time" } #Timer_Delay_Reset.TON(pt := T#1S, et =>)
      R_Coil( #Visual_Test_Approved_PLC )
   END_RUNG
   // the same network as SCL:
   #Timer_Delay_Reset(IN := #Reset_Functional_Test, PT := T#1S);   // TON
   IF #Timer_Delay_Reset.Q THEN #Visual_Test_Approved_PLC := FALSE; END_IF;
END_REGION
END_FUNCTION_BLOCK

DATA_BLOCK "Instance_FB_Digital_Inputs_DB"   // DB101
// stored: AutoNumber false, InstanceOfName FB_Digital_Inputs, InstanceOfType FB
"FB_Digital_Inputs"
   // VAR_INPUT
   //    I_Button_Start_Approve : Bool;
   //    I_Digital_Input_1 : Bool;
   //    I_Digital_Input_2 : Bool;
   //    I_Digital_Input_3 : Bool;
   //    I_Digital_Input_4 : Bool;
   //    I_Digital_Input_5 : Bool;
   // END_VAR
   // VAR_OUTPUT
   //    DB_Button_Start_Approve : Bool;
   //    DB_Digital_Input_1 : Bool;
   //    DB_Digital_Input_2 : Bool;
   //    DB_Digital_Input_3 : Bool;
   //    DB_Digital_Input_4 : Bool;
   //    DB_Digital_Input_5 : Bool;
   // END_VAR
BEGIN
END_DATA_BLOCK

DATA_BLOCK "Instance_FB_Electrical_Current_Test_DB"   // DB106
// stored: AutoNumber false, InstanceOfName FB_Electrical_Current_Test, InstanceOfType FB
"FB_Electrical_Current_Test"
   // VAR_INPUT
   //    Star_Functional_Test : Bool;
   //    Reset_Functional_Test : Bool;
   //    Electrical_Current_Read_UInt : UInt;
   //    In_Test_Parameters : "IO_Device_Test_Parameters";
   // END_VAR
   // VAR_OUTPUT
   //    Electrical_Current_Test_Approved : Bool;
   // END_VAR
   // VAR
   //    Timer_Delay_Read_Current { S7_SetPoint := 'True'} : TON_TIME;
   //    Timer_Delay_Reset { S7_SetPoint := 'True'} : TON_TIME;
   // END_VAR
BEGIN
END_DATA_BLOCK

DATA_BLOCK "Instance_FB_IO_Device_DB"   // DB104
// stored: AutoNumber false, InstanceOfName FB_IO_Device, InstanceOfType FB
"FB_IO_Device"
BEGIN
END_DATA_BLOCK

DATA_BLOCK "Instance_FB_Visual_Test_DB"   // DB107
// stored: AutoNumber false, InstanceOfName FB_Visual_Test, InstanceOfType FB
"FB_Visual_Test"
BEGIN
END_DATA_BLOCK
